// TIA Portal project "Nauriz_uploaded" (V17)

(* hardware
DEVICE "S7-1200 station_1"  S7-1200 Station
   slot 0: "Rack_0"  S7-1200 Rack  Rack  V1.0
   slot 1: "PLC_1"  CPU 1214C DC/DC/DC  6ES7 214-1AG40-0XB0  V4.4
   slot 2: "DI 16x24VDC/DQ 16xRelay_1"  SM 1223 DI16/DQ16 x relay  6ES7 223-1PL32-0XB0  V2.0
   slot 3: "DI 16/DQ 16x24VDC_1"  6ES7 223-1BL32-0XB0  V2.0
   slot 4: "DI 16x24VDC_1"  6ES7 221-1BH32-0XB0  V2.0
   slot 5: "DI 16x24VDC_2"  6ES7 221-1BH32-0XB0  V2.0
   slot 6: "AI 8x13BIT_1"  6ES7 231-4HF32-0XB0  V2.1
   slot 7: "AI 4x13BIT_1"  6ES7 231-4HD32-0XB0  V2.1
   slot 101: "CM 1241 (RS422/485)_1"  6ES7 241-1CH32-0XB0  V2.2
*)

// ===== PLC "PLC_1"  CPU 1214C DC/DC/DC =====

VAR_GLOBAL   // PLC tag table "Default tag table"
   "DIa1.0" AT %I0.0 : Bool;   // Наличие напряжения на основном вводе
   "DIa1.1" AT %I0.1 : Bool;   // Наличие напряжения на резервном вводе
   "DIa1.2" AT %I0.2 : Bool;   // Наличие питания 220 внешних потребителей
   "DIa1.3" AT %I0.3 : Bool;   // Наличие питания 220 собственных нужд
   "DIa1.4" AT %I0.4 : Bool;   // Отключение звука
   "DIa1.5" AT %I0.5 : Bool;   // Стоп АН
   "DIa1.6" AT %I0.6 : Bool;   // Автоматическое управление
   "DIa1.7" AT %I0.7 : Bool;   // Ручное управление
   "DIb1.0" AT %I1.0 : Bool;   // Тест индикации
   "DIb1.1" AT %I1.1 : Bool;   // Затопление
   "DIb1.2" AT %I1.2 : Bool;   // Открытие двери
   "Reserved DIb1.3" AT %I1.3 : Bool;   // ------------------------
   "Reserved DIb1.4" AT %I1.4 : Bool;   // ------------------------
   "Reserved DIb1.5" AT %I1.5 : Bool;   // ------------------------
   "DIa2.0" AT %I8.0 : Bool;   // Авт. выкл. НБ1 включен
   "DIa2.1" AT %I8.1 : Bool;   // Контактор НБ1 включен
   "DIa2.2" AT %I8.2 : Bool;   // Авт. выкл. НБ2 включен
   "DIa2.3" AT %I8.3 : Bool;   // Контактор НБ2 включен
   "DIa2.4" AT %I8.4 : Bool;   // Авт. выкл. НБ3 включен
   "DIa2.5" AT %I8.5 : Bool;   // Контактор НБ3 включен
   "DIa2.6" AT %I8.6 : Bool;   // Авт. выкл. НБ4 включен
   "DIa2.7" AT %I8.7 : Bool;   // Контактор НБ4 включен
   "DIb2.0" AT %I9.0 : Bool;   // Авт. выкл. НБ5 включен
   "DIb2.1" AT %I9.1 : Bool;   // Контактор НБ5 включен
   "DIb2.2" AT %I9.2 : Bool;   // Авт. выкл. НП включен
   "DIb2.3" AT %I9.3 : Bool;   // Контактор НП включен
   "DIb2.4" AT %I9.4 : Bool;   // Авт. выкл. ДР.Н включен
   "DIb2.5" AT %I9.5 : Bool;   // Контактор ДР.Н включен
   "Reserved DIb2.6" AT %I9.6 : Bool;   // ------------------------
   "Reserved DIb2.7" AT %I9.7 : Bool;   // ------------------------
   "DIa3.0" AT %I12.0 : Bool;   // УУС1: Проток
   "DIa3.1" AT %I12.1 : Bool;   // УУС2: Проток
   "DIa3.2" AT %I12.2 : Bool;   // УУС3: Проток
   "DIa3.3" AT %I12.3 : Bool;   // УУС4: Проток
   "DIa3.4" AT %I12.4 : Bool;   // УУС5: Проток
   "DIa3.5" AT %I12.5 : Bool;   // СПЖ1: Проток
   "DIa3.6" AT %I12.6 : Bool;   // Кнопка: Открыть УУД1
   "DIa3.7" AT %I12.7 : Bool;   // АПС: Открыть УУД1
   "DIb3.0" AT %I13.0 : Bool;   // УУС1: Открыт
   "DIb3.1" AT %I13.1 : Bool;   // УУС2: Открыт
   "DIb3.2" AT %I13.2 : Bool;   // УУС3: Открыт
   "DIb3.3" AT %I13.3 : Bool;   // УУС4: Открыт
   "DIb3.4" AT %I13.4 : Bool;   // УУС5: Открыт
   "Reserved DIb3.5" AT %I13.5 : Bool;   // ------------------------
   "Reserved DIb3.6" AT %I13.6 : Bool;   // ------------------------
   "Reserved DIb3.7" AT %I13.7 : Bool;   // ------------------------
   "DIa4.0" AT %I16.0 : Bool;   // Пож. резервуар: Уровень 1
   "DIa4.1" AT %I16.1 : Bool;   // Пож. резервуар: Уровень 2
   "DIa4.2" AT %I16.2 : Bool;   // Пож. резервуар: Уровень 3
   "DIa4.3" AT %I16.3 : Bool;   // Др. приямок: Вкл. ДР.Н
   "DIa4.4" AT %I16.4 : Bool;   // Др. приямок: Верх
   "Reserved DIa4.5" AT %I16.5 : Bool;   // ------------------------
   "Reserved DIa4.6" AT %I16.6 : Bool;   // ------------------------
   "Reserved DIa4.7" AT %I16.7 : Bool;   // ------------------------
   "Reserved DIb4.0" AT %I17.0 : Bool;   // ------------------------
   "Reserved DIb4.1" AT %I17.1 : Bool;   // ------------------------
   "DIb4.2" AT %I17.2 : Bool;   // КР.Ш38 УУС1: Открыт
   "DIb4.3" AT %I17.3 : Bool;   // КР.Ш38 УУС2: Открыт
   "DIb4.4" AT %I17.4 : Bool;   // КР.Ш38 УУС3: Открыт
   "DIb4.5" AT %I17.5 : Bool;   // КР.Ш38 УУС4: Открыт
   "DIb4.6" AT %I17.6 : Bool;   // КР.Ш38 УУС5: Открыт
   "DIb4.7" AT %I17.7 : Bool;   // КР.Ш38 УУД1: Открыт
   "DIa5.0" AT %I20.0 : Bool;   // КР.Ш12 УУС1: Открыт
   "DIa5.1" AT %I20.1 : Bool;   // КР.Ш12 УУС2: Открыт
   "DIa5.2" AT %I20.2 : Bool;   // КР.Ш12 УУС3: Открыт
   "DIa5.3" AT %I20.3 : Bool;   // КР.Ш12 УУС4: Открыт
   "DIa5.4" AT %I20.4 : Bool;   // КР.Ш12 УУС5: Открыт
   "Reserved DIa5.5" AT %I20.5 : Bool;   // ------------------------
   "Reserved DIa5.6" AT %I20.6 : Bool;   // ------------------------
   "Reserved DIa5.7" AT %I20.7 : Bool;   // ------------------------
   "Reserved DIb5.0" AT %I21.0 : Bool;   // ------------------------
   "Reserved DIb5.1" AT %I21.1 : Bool;   // ------------------------
   "Reserved DIb5.2" AT %I21.2 : Bool;   // ------------------------
   "Reserved DIb5.3" AT %I21.3 : Bool;   // ------------------------
   "Reserved DIb5.4" AT %I21.4 : Bool;   // ------------------------
   "Reserved DIb5.5" AT %I21.5 : Bool;   // ------------------------
   "Reserved DIb5.6" AT %I21.6 : Bool;   // ------------------------
   "Reserved DIb5.7" AT %I21.7 : Bool;   // ------------------------
   "AI6.0" AT %IW160 : Int;   // Датчик низкого давления PIS1.1
   "AI6.1" AT %IW162 : Int;   // Датчик низкого давления PIS1.2
   "AI6.2" AT %IW164 : Int;   // Датчик высокого давления PIS2.1
   "AI6.3" AT %IW166 : Int;   // Датчик высокого давления PIS2.2
   "AI6.4" AT %IW168 : Int;   // Датчик давления НБ1
   "AI6.5" AT %IW170 : Int;   // Датчик давления НБ2
   "AI6.6" AT %IW172 : Int;   // Датчик давления НБ3
   "AI6.7" AT %IW174 : Int;   // Датчик давления НБ4
   "AI7.0" AT %IW176 : Int;   // Датчик давления НБ5
   "AI7.1" AT %IW178 : Int;   // Датчик давления УУД1
   "Reserved AI7.2" AT %IW180 : Int;   // ------------------------
   "Reserved AI7.3" AT %IW182 : Int;   // ------------------------
   "DQa1.0" AT %Q0.0 : Bool;   // Пожар
   "DQa1.1" AT %Q0.1 : Bool;   // Пуск
   "DQa1.2" AT %Q0.2 : Bool;   // Неисправность
   "DQa1.3" AT %Q0.3 : Bool;   // Автоматика отключена
   "DQa1.4" AT %Q0.4 : Bool;   // Дежурный режим
   "DQa1.5" AT %Q0.5 : Bool;   // Звуковой сигнал
   "DQa1.6" AT %Q0.6 : Bool;   // СИстема отключена
   "DQa1.7" AT %Q0.7 : Bool;   // Звук отключен
   "DQb1.0" AT %Q1.0 : Bool;   // Наличие ОТВ
   "Reserved DQb1.1" AT %Q1.1 : Bool;   // ------------------------
   "RQa2.0" AT %Q8.0 : Bool;   // Управление НБ1
   "RQa2.1" AT %Q8.1 : Bool;   // Управление НБ2
   "RQa2.2" AT %Q8.2 : Bool;   // Управление НБ3
   "RQa2.3" AT %Q8.3 : Bool;   // Управление НБ4
   "RQa2.4" AT %Q8.4 : Bool;   // Управление НБ5
   "RQa2.5" AT %Q8.5 : Bool;   // Управление НП
   "RQa2.6" AT %Q8.6 : Bool;   // Управление ДР.Н
   "RQa2.7" AT %Q8.7 : Bool;   // Управление УУД1
   "RQb2.0" AT %Q9.0 : Bool;   // Неисправность НБ1
   "RQb2.1" AT %Q9.1 : Bool;   // Неисправность НБ2
   "RQb2.2" AT %Q9.2 : Bool;   // Неисправность НБ3
   "RQb2.3" AT %Q9.3 : Bool;   // Неисправность НБ4
   "RQb2.4" AT %Q9.4 : Bool;   // Неисправность НБ5
   "RQb2.5" AT %Q9.5 : Bool;   // Неисправность НП
   "RQb2.6" AT %Q9.6 : Bool;   // Неисправность ДР.Н
   "Reserved RQb2.7" AT %Q9.7 : Bool;   // ------------------------
   "DQa3.0" AT %Q12.0 : Bool;   // УУС1: Срабатывание
   "DQa3.1" AT %Q12.1 : Bool;   // УУС1: Неисправность
   "DQa3.2" AT %Q12.2 : Bool;   // УУС2: Срабатывание
   "DQa3.3" AT %Q12.3 : Bool;   // УУС2: Неисправность
   "DQa3.4" AT %Q12.4 : Bool;   // УУС3: Срабатывание
   "DQa3.5" AT %Q12.5 : Bool;   // УУС3: Неисправность
   "DQa3.6" AT %Q12.6 : Bool;   // УУС4: Срабатывание
   "DQa3.7" AT %Q12.7 : Bool;   // УУС4: Неисправность
   "DQb3.0" AT %Q13.0 : Bool;   // УУС5: Срабатывание
   "DQb3.1" AT %Q13.1 : Bool;   // УУС5: Неисправность
   "DQb3.2" AT %Q13.2 : Bool;   // УУД1: Открыт
   "DQb3.3" AT %Q13.3 : Bool;   // УУД1: Неисправность
   "Reserved DQb3.4" AT %Q13.4 : Bool;   // ------------------------
   "Reserved DQb3.5" AT %Q13.5 : Bool;   // ------------------------
   "Reserved DQb3.6" AT %Q13.6 : Bool;   // ------------------------
   "Reserved DQb3.7" AT %Q13.7 : Bool;   // ------------------------
   "System_Byte" AT %MB1 : Byte;
   "FirstScan" AT %M1.0 : Bool;
   "DiagStatusUpdate" AT %M1.1 : Bool;
   "AlwaysTRUE" AT %M1.2 : Bool;
   "AlwaysFALSE" AT %M1.3 : Bool;
   "MB_MODE_AUTO" AT %M4001.1 : Bool;
   "MB_MODE_MANUAL" AT %M4001.2 : Bool;
   "MB_MODE_BLOCKED" AT %M4001.3 : Bool;
   "MB_MODE_STANDBY" AT %M4001.4 : Bool;
   "MB_ERROR_ANY" AT %M4003.5 : Bool;
   "MB_ERROR_INLET_PRESSURE_LOW" AT %M4004.0 : Bool;
   "MB_ERROR_PUMP1" AT %M4004.1 : Bool;
   "MB_ERROR_PUMP2" AT %M4004.2 : Bool;
   "MB_ERROR_PUMP3" AT %M4004.3 : Bool;
   "MB_ERROR_PUMP4" AT %M4004.4 : Bool;
   "MB_ERROR_PUMP5" AT %M4004.5 : Bool;
   "MB_ERROR_PRESSURE_SENSOR_PUMP1" AT %M4004.6 : Bool;
   "MB_ERROR_PRESSURE_SENSOR_PUMP2" AT %M4004.7 : Bool;
   "MB_ERROR_PRESSURE_SENSOR_PUMP3" AT %M4005.0 : Bool;
   "MB_ERROR_PRESSURE_SENSOR_PUMP4" AT %M4005.1 : Bool;
   "MB_ERROR_PRESSURE_SENSOR_PUMP5" AT %M4005.2 : Bool;
   "MB_BUTTON_GLOBAL_STOP" AT %M4005.3 : Bool;
   "MB_ERROR_STANDBY_PUMP" AT %M4005.4 : Bool;
   "MB_SENSOR_FLOW_UUS1" AT %M4005.6 : Bool;
   "MB_SENSOR_FLOW_UUS2" AT %M4005.7 : Bool;
   "MB_SENSOR_FLOW_UUS3" AT %M4006.0 : Bool;
   "MB_SENSOR_FLOW_UUS4" AT %M4006.1 : Bool;
   "MB_SENSOR_FLOW_UUS5" AT %M4006.2 : Bool;
   "MB_SIGNAL_OPEN_UUS1" AT %M4006.3 : Bool;
   "MB_SIGNAL_OPEN_UUS2" AT %M4006.4 : Bool;
   "MB_SIGNAL_OPEN_UUS3" AT %M4006.5 : Bool;
   "MB_SIGNAL_OPEN_UUS4" AT %M4006.6 : Bool;
   "MB_SIGNAL_OPEN_UUS5" AT %M4006.7 : Bool;
   "MB_SENSOR_ERROR_UUS1" AT %M4007.0 : Bool;
   "MB_SENSOR_ERROR_UUS2" AT %M4007.1 : Bool;
   "MB_SENSOR_ERROR_UUS3" AT %M4007.2 : Bool;
   "MB_SENSOR_ERROR_UUS4" AT %M4007.3 : Bool;
   "MB_SENSOR_ERROR_UUS5" AT %M4007.4 : Bool;
   "MB_SENSOR_OPEN_KP38.1" AT %M4007.5 : Bool;
   "MB_SENSOR_OPEN_KP38.2" AT %M4007.6 : Bool;
   "MB_SENSOR_OPEN_KP38.3" AT %M4007.7 : Bool;
   "MB_SENSOR_OPEN_KP38.4" AT %M4008.0 : Bool;
   "MB_SENSOR_OPEN_KP38.5" AT %M4008.1 : Bool;
   "MB_SENSOR_OPEN_KP38.6" AT %M4008.2 : Bool;
   "MB_STATE_380_MAIN" AT %M4001.5 : Bool;
   "MB_STATE_380_BACKUP" AT %M4001.6 : Bool;
   "MB_STATE_220_INNER" AT %M4001.7 : Bool;
   "MB_STATE_220_OUTER" AT %M4002.0 : Bool;
   "MB_STATE_DOOR_OPENED" AT %M4002.1 : Bool;
   "MB_ERROR_UNDERWATER" AT %M4002.3 : Bool;
   "MB_ERROR_NO_WATER" AT %M4002.4 : Bool;
   "MB_ERROR_NO_WATER_FIRE" AT %M4002.5 : Bool;
   "MB_ERROR_GLOBAL" AT %M4003.1 : Bool;
   "MB_ERROR_UUS" AT %M4003.2 : Bool;
   "MB_ERROR_UUS_ANY" AT %M4003.3 : Bool;
   "MB_ERROR_PUMPS" AT %M4003.6 : Bool;
   "MB_ERROR_BALL_VALVE_ANY" AT %M4003.7 : Bool;
   "MB_SIGNAL_FIRE" AT %M4002.2 : Bool;
   "MB_SENSOR_PRESSURE_PUMP1" AT %MD4012 : Real;
   "MB_SENSOR_PRESSURE_PUMP2" AT %MD4016 : Real;
   "MB_SENSOR_PRESSURE_PUMP3" AT %MD4020 : Real;
   "MB_SENSOR_PRESSURE_PUMP4" AT %MD4024 : Real;
   "MB_SENSOR_PRESSURE_PUMP5" AT %MD4028 : Real;
   "MB_SENSOR_INDICATION_PRESSURE_LOW" AT %MD4032 : Real;
   "MB_SENSOR_INDICATION_PRESSURE_HIGH" AT %MD4036 : Real;
   "MB_STATE_WORK_PUMP1" AT %M4009.0 : Bool;
   "MB_STATE_WORK_PUMP2" AT %M4009.1 : Bool;
   "MB_STATE_WORK_PUMP3" AT %M4009.2 : Bool;
   "MB_STATE_WORK_PUMP4" AT %M4009.3 : Bool;
   "MB_STATE_WORK_PUMP5" AT %M4009.4 : Bool;
   "MB_STATE_WORK_STANDBY_PUMP" AT %M4009.5 : Bool;
   "MB_STATE_WORK_ANY_PUMP" AT %M4009.6 : Bool;
   "MB_ERROR_CONNECTION_LOST" AT %M4010.5 : Bool;
   "MB_BUTTON_START_KPPU" AT %M4000.2 : Bool;
   "MB_BUTTON_STOP_KPPU" AT %M4000.1 : Bool;
   "MB_BUTTON_UUD_OPEN_KPPU" AT %M4000.3 : Bool;
   "MB_WATER_LEVEL_FULL" AT %M4002.6 : Bool;
   "MB_SIGNAL_NEED_REPLENISH_1" AT %M4002.7 : Bool;
   "MB_SIGNAL_NEED_REPLENISH_2" AT %M4003.0 : Bool;
   "MB_ERROR_UUD1" AT %M4003.4 : Bool;
   "MB_ERROR_DRAIN_PUMP" AT %M4005.5 : Bool;
   "MB_STATE_WORK_DRAIN_PUMP" AT %M4009.7 : Bool;
   "MB_Sensor_water_level_1" AT %M4010.0 : Bool;
   "MB_Sensor_water_level_2" AT %M4010.1 : Bool;
   "MB_Sensor_water_level_3" AT %M4010.2 : Bool;
   "MB_Sensor_drain_work" AT %M4010.3 : Bool;
   "MB_Sensor_drain_overflow" AT %M4010.4 : Bool;
   "MB_SENSOR_OPEN_KP12.1" AT %M4008.3 : Bool;
   "MB_SENSOR_OPEN_KP12.2" AT %M4008.4 : Bool;
   "MB_SENSOR_OPEN_KP12.3" AT %M4008.5 : Bool;
   "MB_SENSOR_OPEN_KP12.4" AT %M4008.6 : Bool;
   "MB_SENSOR_OPEN_KP12.5" AT %M4008.7 : Bool;
   "Commload_done" AT %M900.0 : Bool;
   "Master_reading_done" AT %M900.1 : Bool;
   "Master_writing_done" AT %M900.2 : Bool;
   "Master_reading_error" AT %M900.3 : Bool;
   "Master_writing_error" AT %M900.4 : Bool;
   "Master_read" AT %M900.5 : Bool;
   "Master_write" AT %M900.6 : Bool;
   "Error_connection_lost" AT %M900.7 : Bool;
   "WriteHoldingRegister_00" AT %MW4002 : Word;
   "WriteHoldingRegister_01" AT %MW4004 : Word;
   "WriteHoldingRegister_02" AT %MW4006 : Word;
   "WriteHoldingRegister_03" AT %MW4008 : Word;
   "WriteHoldingRegister_04" AT %MW4010 : Word;
   "WriteHoldingRegister_05" AT %MW4012 : Word;
   "WriteHoldingRegister_06" AT %MW4014 : Word;
   "WriteHoldingRegister_07" AT %MW4016 : Word;
   "WriteHoldingRegister_08" AT %MW4018 : Word;
   "WriteHoldingRegister_09" AT %MW4020 : Word;
   "WriteHoldingRegister_10" AT %MW4022 : Word;
   "WriteHoldingRegister_11" AT %MW4024 : Word;
   "WriteHoldingRegister_12" AT %MW4026 : Word;
   "WriteHoldingRegister_13" AT %MW4028 : Word;
   "WriteHoldingRegister_14" AT %MW4030 : Word;
   "WriteHoldingRegister_15" AT %MW4032 : Word;
   "WriteHoldingRegister_16" AT %MW4034 : Word;
   "WriteHoldingRegister_18" AT %MW4038 : Word;
   "WriteHoldingRegister_19" AT %MW4040 : Word;
   "WriteHoldingRegister_20" AT %MW4042 : Word;
   "WriteHoldingRegister_22" AT %MW4046 : Word;
   "WriteHoldingRegister_23" AT %MW4048 : Word;
   "WriteHoldingRegister_24" AT %MW4050 : Word;
   "WriteHoldingRegister_25" AT %MW4052 : Word;
   "WriteHoldingRegister_26" AT %MW4054 : Word;
   "WriteHoldingRegister_27" AT %MW4056 : Word;
   "WriteHoldingRegister_28" AT %MW4058 : Word;
   "WriteHoldingRegister_29" AT %MW4060 : Word;
   "WriteHoldingRegister_30" AT %MW4062 : Word;
   "WriteHoldingRegister_31" AT %MW4064 : Word;
   "WriteHoldingRegister_32" AT %MW4066 : Word;
   "WriteHoldingRegister_33" AT %MW4068 : Word;
   "WriteHoldingRegister_34" AT %MW4070 : Word;
   "WriteHoldingRegister_35" AT %MW4072 : Word;
   "WriteHoldingRegister_36" AT %MW4074 : Word;
   "WriteHoldingRegister_37" AT %MW4076 : Word;
   "WriteHoldingRegister_38" AT %MW4078 : Word;
   "ReadHolding" AT %MW4000 : Word;
   "WriteHoldingRegister_17" AT %MW4036 : Word;
   "WriteHoldingRegister_21" AT %MW4044 : Word;
   "HMI_MODE_AUTO" AT %M600.0 : Bool;
   "HMI_MODE_MANUAL" AT %M600.1 : Bool;
   "HMI_MODE_BLOCKED" AT %M600.2 : Bool;
   "HMI_MODE_STANDBY" AT %M600.3 : Bool;
   "HMI_ERROR_ANY" AT %M600.4 : Bool;
   "HMI_ERROR_INLET_PRESSURE_LOW" AT %M600.5 : Bool;
   "HMI_ERROR_PUMP1" AT %M600.6 : Bool;
   "HMI_ERROR_PUMP2" AT %M600.7 : Bool;
   "HMI_ERROR_PUMP3" AT %M601.0 : Bool;
   "HMI_ERROR_PUMP4" AT %M601.1 : Bool;
   "HMI_ERROR_PUMP5" AT %M601.2 : Bool;
   "HMI_ERROR_PRESSURE_SENSOR_PUMP1" AT %M601.3 : Bool;
   "HMI_ERROR_PRESSURE_SENSOR_PUMP2" AT %M601.4 : Bool;
   "HMI_ERROR_PRESSURE_SENSOR_PUMP3" AT %M601.5 : Bool;
   "HMI_ERROR_PRESSURE_SENSOR_PUMP4" AT %M601.6 : Bool;
   "HMI_ERROR_PRESSURE_SENSOR_PUMP5" AT %M601.7 : Bool;
   "HMI_BUTTON_GLOBAL_STOP" AT %M602.0 : Bool;
   "HMI_ERROR_STANDBY_PUMP" AT %M602.1 : Bool;
   "HMI_SENSOR_FLOW_UUS1" AT %M602.2 : Bool;
   "HMI_SENSOR_FLOW_UUS2" AT %M602.3 : Bool;
   "HMI_SENSOR_FLOW_UUS3" AT %M602.4 : Bool;
   "HMI_SENSOR_FLOW_UUS4" AT %M602.5 : Bool;
   "HMI_SENSOR_FLOW_UUS5" AT %M602.6 : Bool;
   "HMI_SIGNAL_OPEN_UUS1" AT %M602.7 : Bool;
   "HMI_SIGNAL_OPEN_UUS2" AT %M603.0 : Bool;
   "HMI_SIGNAL_OPEN_UUS3" AT %M603.1 : Bool;
   "HMI_SIGNAL_OPEN_UUS4" AT %M603.2 : Bool;
   "HMI_SIGNAL_OPEN_UUS5" AT %M603.3 : Bool;
   "HMI_SENSOR_ERROR_UUS1" AT %M603.4 : Bool;
   "HMI_SENSOR_ERROR_UUS2" AT %M603.5 : Bool;
   "HMI_SENSOR_ERROR_UUS3" AT %M603.6 : Bool;
   "HMI_SENSOR_ERROR_UUS4" AT %M603.7 : Bool;
   "HMI_SENSOR_ERROR_UUS5" AT %M604.0 : Bool;
   "HMI_SENSOR_OPEN_KP38.1" AT %M604.1 : Bool;
   "HMI_SENSOR_OPEN_KP38.2" AT %M604.2 : Bool;
   "HMI_SENSOR_OPEN_KP38.3" AT %M604.3 : Bool;
   "HMI_SENSOR_OPEN_KP38.4" AT %M604.4 : Bool;
   "HMI_SENSOR_OPEN_KP38.5" AT %M604.5 : Bool;
   "HMI_SENSOR_OPEN_KP38.6" AT %M604.6 : Bool;
   "HMI_STATE_380_MAIN" AT %M604.7 : Bool;
   "HMI_STATE_380_BACKUP" AT %M605.0 : Bool;
   "HMI_STATE_220_INNER" AT %M605.1 : Bool;
   "HMI_STATE_220_OUTER" AT %M605.2 : Bool;
   "HMI_STATE_DOOR_OPENED" AT %M605.3 : Bool;
   "HMI_ERROR_UNDERWATER" AT %M605.4 : Bool;
   "HMI_ERROR_NO_WATER" AT %M605.5 : Bool;
   "HMI_ERROR_NO_WATER_FIRE" AT %M605.6 : Bool;
   "HMI_ERROR_GLOBAL" AT %M605.7 : Bool;
   "HMI_ERROR_UUS" AT %M606.0 : Bool;
   "HMI_ERROR_UUS_ANY" AT %M606.1 : Bool;
   "HMI_ERROR_PUMPS" AT %M606.2 : Bool;
   "HMI_ERROR_BALL_VALVE_ANY" AT %M606.3 : Bool;
   "HMI_SIGNAL_FIRE" AT %M606.4 : Bool;
   "HMI_SENSOR_PRESSURE_PUMP1" AT %MD610 : Real;
   "HMI_SENSOR_PRESSURE_PUMP2" AT %MD614 : Real;
   "HMI_SENSOR_PRESSURE_PUMP3" AT %MD618 : Real;
   "HMI_SENSOR_PRESSURE_PUMP4" AT %MD622 : Real;
   "HMI_SENSOR_PRESSURE_PUMP5" AT %MD626 : Real;
   "HMI_SENSOR_INDICATION_PRESSURE_LOW" AT %MD630 : Real;
   "HMI_SENSOR_INDICATION_PRESSURE_HIGH" AT %MD634 : Real;
   "HMI_STATE_WORK_PUMP1" AT %M606.5 : Bool;
   "HMI_STATE_WORK_PUMP2" AT %M606.6 : Bool;
   "HMI_STATE_WORK_PUMP3" AT %M606.7 : Bool;
   "HMI_STATE_WORK_PUMP4" AT %M607.0 : Bool;
   "HMI_STATE_WORK_PUMP5" AT %M607.1 : Bool;
   "HMI_STATE_WORK_STANDBY_PUMP" AT %M607.2 : Bool;
   "HMI_STATE_WORK_ANY_PUMP" AT %M607.3 : Bool;
   "HMI_ERROR_CONNECTION_LOST" AT %M607.4 : Bool;
   "HMI_BUTTON_START_KPPU" AT %M607.5 : Bool;
   "HMI_BUTTON_STOP_KPPU" AT %M607.6 : Bool;
   "HMI_BUTTON_UUD_OPEN_KPPU" AT %M607.7 : Bool;
   "HMI_WATER_LEVEL_FULL" AT %M608.0 : Bool;
   "HMI_SIGNAL_NEED_REPLENISH_1" AT %M608.1 : Bool;
   "HMI_SIGNAL_NEED_REPLENISH_2" AT %M608.2 : Bool;
   "HMI_ERROR_UUD1" AT %M608.3 : Bool;
   "HMI_ERROR_DRAIN_PUMP" AT %M608.4 : Bool;
   "HMI_STATE_WORK_DRAIN_PUMP" AT %M608.5 : Bool;
   "HMI_Sensor_water_level_1" AT %M608.6 : Bool;
   "HMI_Sensor_water_level_2" AT %M608.7 : Bool;
   "HMI_Sensor_water_level_3" AT %M609.0 : Bool;
   "HMI_Sensor_drain_work" AT %M609.1 : Bool;
   "HMI_Sensor_drain_overflow" AT %M609.2 : Bool;
   "HMI_SENSOR_OPEN_KP12.1" AT %M609.3 : Bool;
   "HMI_SENSOR_OPEN_KP12.2" AT %M609.4 : Bool;
   "HMI_SENSOR_OPEN_KP12.3" AT %M609.5 : Bool;
   "HMI_SENSOR_OPEN_KP12.4" AT %M609.6 : Bool;
   "HMI_SENSOR_OPEN_KP12.5" AT %M609.7 : Bool;
END_VAR

DATA_BLOCK "Ball_valves_data"   // DB1
{ S7_Optimized_Access := 'TRUE' }
VERSION : 0.1
   VAR
      SENSOR_KR38_open : Array[1..6] of Bool;
      SENSOR_KR12_open : Array[1..5] of Bool;
      SENSOR_ERROR_KR38 : Array[1..6] of Bool;
   END_VAR
BEGIN
END_DATA_BLOCK

DATA_BLOCK "Section_valves_data"   // DB2
{ S7_Optimized_Access := 'TRUE' }
VERSION : 0.1
   VAR
      SENSOR_flow_UUS : Array[1..5] of Bool;
      SENSOR_ERROR_UUS : Array[1..5] of Bool;
      SENSOR_open_UUS : Array[1..5] of Bool;
      SENSOR_ERROR_UUD1 : Bool;
      SENSOR_open_UUD1 : Bool;
      SENSOR_FALSE_UUD1 : Bool;
   END_VAR
BEGIN
END_DATA_BLOCK

DATA_BLOCK "Global"   // DB47
{ S7_Optimized_Access := 'TRUE' }
VERSION : 0.1
   VAR
      MODE_auto : Bool;
      MODE_manual : Bool;
      MODE_blocked : Bool;
      MODE_standby : Bool;
      BUTTON_Global_Stop : Bool;
      BUTTON_Sound_Off : Bool;
      BUTTON_Led_Test : Bool;
      BUTTON_UUD1_Open : Bool;
      STATE_380_main : Bool;
      STATE_380_backup : Bool;
      STATE_220_inner : Bool;
      STATE_220_outer : Bool;
      STATE_door_opened : Bool;
      ERROR_underwater : Bool;
      ERROR_no_water : Bool;
      ERROR_no_water_fire : Bool;
      ERROR_global : Bool;
      ERROR_UUS : Bool;
      ERROR_UUS_any : Bool;
      ERROR_any : Bool;
      ERROR_PUMPS : Bool;
      SIGNAL_fire : Bool;
      "SENSOR_low_pressure_PIS1.1" : Real;
      "SENSOR_low_pressure_PIS1.2" : Real := 0.0;
      "SENSOR_high_pressure_PIS2.1" : Real := 0.0;
      "SENSOR_high_pressure_PIS2.2" : Real := 0.0;
      SENSOR_high_pressure_pump_1 : Real := 0.0;
      SENSOR_high_pressure_pump_2 : Real := 0.0;
      SENSOR_high_pressure_pump_3 : Real := 0.0;
      SENSOR_high_pressure_pump_4 : Real := 0.0;
      SENSOR_high_pressure_pump_5 : Real := 0.0;
      SENSOR_high_pressure_UUD1 : Real;
      INDICATION_low_pressure : Real := 0.0;
      INDICATION_high_pressure : Real := 0.0;
      ERROR_main_ball_valves : Bool;
      ERROR_ball_valve_any : Bool;
      ERROR_inlet_pressure_low : Bool;
      SIGNAL_first_pump_has_started : Bool;
      Start_standby_pump : Bool;
      Secret_condition : Bool := false;
      Sensor_water_level_1 : Bool;
      Sensor_water_level_2 : Bool;
      Sensor_water_level_3 : Bool;
      Sensor_drain_work : Bool;
      Sensor_drain_overflow : Bool;
      AI_sensors_error : Array[1..4] of Bool;
   END_VAR
BEGIN
END_DATA_BLOCK

DATA_BLOCK "AI_Sensor_high_pressure_UUD1"   // DB58
{ S7_Optimized_Access := 'TRUE' }
VERSION : 0.1
// stored: InstanceOfName AI_Sensor
"AI_Sensor"
BEGIN
END_DATA_BLOCK

DATA_BLOCK "Sound_DB"   // DB59
{ S7_Optimized_Access := 'TRUE' }
VERSION : 0.1
// stored: InstanceOfName Sound_PTO
"Sound_PTO"
BEGIN
END_DATA_BLOCK

DATA_BLOCK "Preset_values"   // DB69
{ S7_Optimized_Access := 'TRUE' }
VERSION : 0.1
   VAR
      DI_timer_delay_time_superfast : Time := T#0.2s;
      DI_timer_delay_time_fast : Time := T#0.5s;
      DI_timer_delay_time_regular : Time := T#1s;
      DI_timer_delay_time_slow : Time := T#3s;
      DI_timer_delay_time_superslow : Time := T#5s;
      DI_timer_delay_time_gate_valve : Time := T#30s;
      Pressure_stanby_low : Real := 2.29;
      Pressure_stanby_pump_on : Real := 2.3;
      Pressure_stanby_pump_stop : Real := 2.5;
      Pressure_cascade_start : Real := 7.5;
      Pressure_cascade_stop : Real := 9.0;
      Pressure_pump_is_ok : Real := 10.0;
      Timer_cascade_start : Time := T#25s;
      Pump_error_time_by_pressure : Time := T#60s;
   END_VAR
BEGIN
END_DATA_BLOCK

DATA_BLOCK "Water_control"   // DB71
{ S7_Optimized_Access := 'TRUE' }
VERSION : 0.1
   VAR
      Water_level_full : Bool;
      Signal_need_replenish_1 : Bool;
      Signal_need_replenish_2 : Bool;
   END_VAR
BEGIN
END_DATA_BLOCK

DATA_BLOCK "Cascade_start_stop_DB"   // DB72
{ S7_Optimized_Access := 'TRUE' }
VERSION : 0.1
// stored: InstanceOfName Cascade_start_stop
"Cascade_start_stop"
BEGIN
END_DATA_BLOCK

DATA_BLOCK "Pumps_data"   // DB73
{ S7_Optimized_Access := 'TRUE' }
VERSION : 0.1
   VAR
      State_switch_pump : Array[1..5] of Bool;
      Error_pump : Array[1..5] of Bool;
      State_starter_pump : Array[1..5] of Bool;
      State_work_pump : Array[1..5] of Bool;
      Pumps : Array[1..5] of Int;
      Pump_sensor_error : Array[1..5] of Bool;
      State_switch_standby_pump : Bool;
      Error_any_pump : Bool;
      Error_standby_pump : Bool;
      State_starter_standby_pump : Bool;
      State_work_standby_pump : Bool;
      State_work_any_pump : Bool;
      State_switch_drain_pump : Bool;
      State_starter_drain_pump : Bool;
      Error_drain_pump : Bool;
      State_work_drain_pump : Bool;
   END_VAR
BEGIN
END_DATA_BLOCK

DATA_BLOCK "Data_push_to_MODBUS_DB"   // DB85
{ S7_Optimized_Access := 'TRUE' }
VERSION : 0.1
// stored: InstanceOfName Data_push_to_MODBUS
"Data_push_to_MODBUS"
BEGIN
END_DATA_BLOCK

DATA_BLOCK "Data_push_to_HMI_DB"   // DB87
{ S7_Optimized_Access := 'TRUE' }
VERSION : 0.1
// stored: InstanceOfName Data_push_to_HMI
"Data_push_to_HMI"
BEGIN
END_DATA_BLOCK

DATA_BLOCK "User_Defined"   // DB100
{ S7_Optimized_Access := 'TRUE' }
VERSION : 0.1
   VAR
      Pressure_stanby_low : Real := 2.29;
      Pressure_stanby_pump_on : Real := 2.3;
      Pressure_stanby_pump_stop : Real := 2.5;
      Pressure_cascade_start : Real := 7.5;
      Pressure_cascade_stop : Real := 9.0;
      Pressure_pump_is_ok : Real := 10.0;
      Timer_cascade_start : Time := T#25s;
      Timer_standby_pump : Time := T#40ms;
      Pump_error_time_by_pressure : Time := T#60s;
   END_VAR
BEGIN
END_DATA_BLOCK

// folder: AI_db

DATA_BLOCK "AI_Sensor_low_pressure_PIS1.1"   // DB43
{ S7_Optimized_Access := 'TRUE' }
VERSION : 0.1
// stored: InstanceOfName AI_Sensor
"AI_Sensor"
BEGIN
END_DATA_BLOCK

DATA_BLOCK "AI_Sensor_low_pressure_PIS1.2"   // DB44
{ S7_Optimized_Access := 'TRUE' }
VERSION : 0.1
// stored: InstanceOfName AI_Sensor
"AI_Sensor"
BEGIN
END_DATA_BLOCK

DATA_BLOCK "AI_Sensor_high_pressure_PIS2.1"   // DB45
{ S7_Optimized_Access := 'TRUE' }
VERSION : 0.1
// stored: InstanceOfName AI_Sensor
"AI_Sensor"
BEGIN
END_DATA_BLOCK

DATA_BLOCK "AI_Sensor_high_pressure_PIS2.2"   // DB46
{ S7_Optimized_Access := 'TRUE' }
VERSION : 0.1
// stored: InstanceOfName AI_Sensor
"AI_Sensor"
BEGIN
END_DATA_BLOCK

DATA_BLOCK "AI_Sensor_high_pressure_pump_1"   // DB48
{ S7_Optimized_Access := 'TRUE' }
VERSION : 0.1
// stored: InstanceOfName AI_Sensor
"AI_Sensor"
BEGIN
END_DATA_BLOCK

DATA_BLOCK "AI_Sensor_high_pressure_pump_2"   // DB49
{ S7_Optimized_Access := 'TRUE' }
VERSION : 0.1
// stored: InstanceOfName AI_Sensor
"AI_Sensor"
BEGIN
END_DATA_BLOCK

DATA_BLOCK "AI_Sensor_high_pressure_pump_3"   // DB50
{ S7_Optimized_Access := 'TRUE' }
VERSION : 0.1
// stored: InstanceOfName AI_Sensor
"AI_Sensor"
BEGIN
END_DATA_BLOCK

DATA_BLOCK "AI_Sensor_high_pressure_pump_4"   // DB51
{ S7_Optimized_Access := 'TRUE' }
VERSION : 0.1
// stored: InstanceOfName AI_Sensor
"AI_Sensor"
BEGIN
END_DATA_BLOCK

DATA_BLOCK "AI_Sensor_high_pressure_pump_5"   // DB52
{ S7_Optimized_Access := 'TRUE' }
VERSION : 0.1
// stored: InstanceOfName AI_Sensor
"AI_Sensor"
BEGIN
END_DATA_BLOCK

DATA_BLOCK "AI_Redundancy_low_pressure"   // DB56
{ S7_Optimized_Access := 'TRUE' }
VERSION : 0.1
// stored: InstanceOfName AI_Redundancy
"AI_Redundancy"
BEGIN
END_DATA_BLOCK

DATA_BLOCK "AI_Redundancy_high_pressure"   // DB57
{ S7_Optimized_Access := 'TRUE' }
VERSION : 0.1
// stored: InstanceOfName AI_Redundancy
"AI_Redundancy"
BEGIN
END_DATA_BLOCK

// folder: DI_db

DATA_BLOCK "State_380_main"   // DB3
{ S7_Optimized_Access := 'TRUE' }
VERSION : 0.1
// stored: InstanceOfName DI_Single
"DI_Single"
BEGIN
END_DATA_BLOCK

DATA_BLOCK "State_380_backup"   // DB4
{ S7_Optimized_Access := 'TRUE' }
VERSION : 0.1
// stored: InstanceOfName DI_Single
"DI_Single"
BEGIN
END_DATA_BLOCK

DATA_BLOCK "State_220_outer"   // DB5
{ S7_Optimized_Access := 'TRUE' }
VERSION : 0.1
// stored: InstanceOfName DI_Single
"DI_Single"
BEGIN
END_DATA_BLOCK

DATA_BLOCK "State_220_inner"   // DB6
{ S7_Optimized_Access := 'TRUE' }
VERSION : 0.1
// stored: InstanceOfName DI_Single
"DI_Single"
BEGIN
END_DATA_BLOCK

DATA_BLOCK "State_Mode_Auto"   // DB7
{ S7_Optimized_Access := 'TRUE' }
VERSION : 0.1
// stored: InstanceOfName DI_Single
"DI_Single"
BEGIN
END_DATA_BLOCK

DATA_BLOCK "State_mode_manual"   // DB8
{ S7_Optimized_Access := 'TRUE' }
VERSION : 0.1
// stored: InstanceOfName DI_Single
"DI_Single"
BEGIN
END_DATA_BLOCK

DATA_BLOCK "State_underwater"   // DB9
{ S7_Optimized_Access := 'TRUE' }
VERSION : 0.1
// stored: InstanceOfName DI_Single
"DI_Single"
BEGIN
END_DATA_BLOCK

DATA_BLOCK "State_door_opened"   // DB10
{ S7_Optimized_Access := 'TRUE' }
VERSION : 0.1
// stored: InstanceOfName DI_Single
"DI_Single"
BEGIN
END_DATA_BLOCK

DATA_BLOCK "Button_UUD1_Open"   // DB11
{ S7_Optimized_Access := 'TRUE' }
VERSION : 0.1
// stored: InstanceOfName DI_Single
"DI_Single"
BEGIN
END_DATA_BLOCK

DATA_BLOCK "Button_sound_off"   // DB12
{ S7_Optimized_Access := 'TRUE' }
VERSION : 0.1
// stored: InstanceOfName DI_Single
"DI_Single"
BEGIN
END_DATA_BLOCK

DATA_BLOCK "Button_global_stop"   // DB13
{ S7_Optimized_Access := 'TRUE' }
VERSION : 0.1
// stored: InstanceOfName DI_Single
"DI_Single"
BEGIN
END_DATA_BLOCK

DATA_BLOCK "Button_led_test"   // DB14
{ S7_Optimized_Access := 'TRUE' }
VERSION : 0.1
// stored: InstanceOfName DI_Single
"DI_Single"
BEGIN
END_DATA_BLOCK

DATA_BLOCK "State_pump_1"   // DB15
{ S7_Optimized_Access := 'TRUE' }
VERSION : 0.1
// stored: InstanceOfName DI_Single
"DI_Single"
BEGIN
END_DATA_BLOCK

DATA_BLOCK "State_pump_2"   // DB16
{ S7_Optimized_Access := 'TRUE' }
VERSION : 0.1
// stored: InstanceOfName DI_Single
"DI_Single"
BEGIN
END_DATA_BLOCK

DATA_BLOCK "State_pump_3"   // DB17
{ S7_Optimized_Access := 'TRUE' }
VERSION : 0.1
// stored: InstanceOfName DI_Single
"DI_Single"
BEGIN
END_DATA_BLOCK

DATA_BLOCK "State_pump_4"   // DB18
{ S7_Optimized_Access := 'TRUE' }
VERSION : 0.1
// stored: InstanceOfName DI_Single
"DI_Single"
BEGIN
END_DATA_BLOCK

DATA_BLOCK "State_pump_5"   // DB19
{ S7_Optimized_Access := 'TRUE' }
VERSION : 0.1
// stored: InstanceOfName DI_Single
"DI_Single"
BEGIN
END_DATA_BLOCK

DATA_BLOCK "State_drain_pump"   // DB20
{ S7_Optimized_Access := 'TRUE' }
VERSION : 0.1
// stored: InstanceOfName DI_Single
"DI_Single"
BEGIN
END_DATA_BLOCK

DATA_BLOCK "State_starter_drain_pump"   // DB21
{ S7_Optimized_Access := 'TRUE' }
VERSION : 0.1
// stored: InstanceOfName DI_Single
"DI_Single"
BEGIN
END_DATA_BLOCK

DATA_BLOCK "Sensor_UUS1_Open"   // DB22
{ S7_Optimized_Access := 'TRUE' }
VERSION : 0.1
// stored: InstanceOfName DI_Single
"DI_Single"
BEGIN
END_DATA_BLOCK

DATA_BLOCK "State_standby_pump"   // DB23
{ S7_Optimized_Access := 'TRUE' }
VERSION : 0.1
// stored: InstanceOfName DI_Single
"DI_Single"
BEGIN
END_DATA_BLOCK

DATA_BLOCK "State_starter_pump_1"   // DB24
{ S7_Optimized_Access := 'TRUE' }
VERSION : 0.1
// stored: InstanceOfName DI_Single
"DI_Single"
BEGIN
END_DATA_BLOCK

DATA_BLOCK "State_starter_pump_2"   // DB25
{ S7_Optimized_Access := 'TRUE' }
VERSION : 0.1
// stored: InstanceOfName DI_Single
"DI_Single"
BEGIN
END_DATA_BLOCK

DATA_BLOCK "State_starter_pump_3"   // DB26
{ S7_Optimized_Access := 'TRUE' }
VERSION : 0.1
// stored: InstanceOfName DI_Single
"DI_Single"
BEGIN
END_DATA_BLOCK

DATA_BLOCK "State_starter_pump_4"   // DB27
{ S7_Optimized_Access := 'TRUE' }
VERSION : 0.1
// stored: InstanceOfName DI_Single
"DI_Single"
BEGIN
END_DATA_BLOCK

DATA_BLOCK "State_starter_pump_5"   // DB28
{ S7_Optimized_Access := 'TRUE' }
VERSION : 0.1
// stored: InstanceOfName DI_Single
"DI_Single"
BEGIN
END_DATA_BLOCK

DATA_BLOCK "Sensor_UUS2_open"   // DB29
{ S7_Optimized_Access := 'TRUE' }
VERSION : 0.1
// stored: InstanceOfName DI_Single
"DI_Single"
BEGIN
END_DATA_BLOCK

DATA_BLOCK "Sensor_UUS3_open"   // DB30
{ S7_Optimized_Access := 'TRUE' }
VERSION : 0.1
// stored: InstanceOfName DI_Single
"DI_Single"
BEGIN
END_DATA_BLOCK

DATA_BLOCK "Sensor_UUS4_open"   // DB31
{ S7_Optimized_Access := 'TRUE' }
VERSION : 0.1
// stored: InstanceOfName DI_Single
"DI_Single"
BEGIN
END_DATA_BLOCK

DATA_BLOCK "State_starter_standby_pump"   // DB32
{ S7_Optimized_Access := 'TRUE' }
VERSION : 0.1
// stored: InstanceOfName DI_Single
"DI_Single"
BEGIN
END_DATA_BLOCK

DATA_BLOCK "Sensor_flow_UUS1"   // DB33
{ S7_Optimized_Access := 'TRUE' }
VERSION : 0.1
// stored: InstanceOfName DI_Single
"DI_Single"
BEGIN
END_DATA_BLOCK

DATA_BLOCK "Sensor_flow_UUS2"   // DB34
{ S7_Optimized_Access := 'TRUE' }
VERSION : 0.1
// stored: InstanceOfName DI_Single
"DI_Single"
BEGIN
END_DATA_BLOCK

DATA_BLOCK "Sensor_flow_UUS3"   // DB35
{ S7_Optimized_Access := 'TRUE' }
VERSION : 0.1
// stored: InstanceOfName DI_Single
"DI_Single"
BEGIN
END_DATA_BLOCK

DATA_BLOCK "Sensor_flow_UUS4"   // DB36
{ S7_Optimized_Access := 'TRUE' }
VERSION : 0.1
// stored: InstanceOfName DI_Single
"DI_Single"
BEGIN
END_DATA_BLOCK

DATA_BLOCK "Sensor_flow_UUS5"   // DB37
{ S7_Optimized_Access := 'TRUE' }
VERSION : 0.1
// stored: InstanceOfName DI_Single
"DI_Single"
BEGIN
END_DATA_BLOCK

DATA_BLOCK "Sensor_UUS5_open"   // DB38
{ S7_Optimized_Access := 'TRUE' }
VERSION : 0.1
// stored: InstanceOfName DI_Single
"DI_Single"
BEGIN
END_DATA_BLOCK

DATA_BLOCK "Sensor_KR38.1_open"   // DB39
{ S7_Optimized_Access := 'TRUE' }
VERSION : 0.1
// stored: InstanceOfName DI_Single
"DI_Single"
BEGIN
END_DATA_BLOCK

DATA_BLOCK "Sensor_KR38.2_open"   // DB40
{ S7_Optimized_Access := 'TRUE' }
VERSION : 0.1
// stored: InstanceOfName DI_Single
"DI_Single"
BEGIN
END_DATA_BLOCK

DATA_BLOCK "Sensor_KR38.3_open"   // DB41
{ S7_Optimized_Access := 'TRUE' }
VERSION : 0.1
// stored: InstanceOfName DI_Single
"DI_Single"
BEGIN
END_DATA_BLOCK

DATA_BLOCK "Sensor_KR38.4_open"   // DB42
{ S7_Optimized_Access := 'TRUE' }
VERSION : 0.1
// stored: InstanceOfName DI_Single
"DI_Single"
BEGIN
END_DATA_BLOCK

DATA_BLOCK "Sensor_water_level_3"   // DB53
{ S7_Optimized_Access := 'TRUE' }
VERSION : 0.1
// stored: InstanceOfName DI_Single
"DI_Single"
BEGIN
END_DATA_BLOCK

DATA_BLOCK "Sensor_drain_work"   // DB54
{ S7_Optimized_Access := 'TRUE' }
VERSION : 0.1
// stored: InstanceOfName DI_Single
"DI_Single"
BEGIN
END_DATA_BLOCK

DATA_BLOCK "Sensor_drain_overflow"   // DB55
{ S7_Optimized_Access := 'TRUE' }
VERSION : 0.1
// stored: InstanceOfName DI_Single
"DI_Single"
BEGIN
END_DATA_BLOCK

DATA_BLOCK "Standby_Pump/Compressor_Error_DB"   // DB60
{ S7_Optimized_Access := 'TRUE' }
VERSION : 0.1
// stored: InstanceOfName Standby_Pump/Compressor_Error
"Standby_Pump/Compressor_Error"
BEGIN
END_DATA_BLOCK

DATA_BLOCK "Pump_Error_1"   // DB61
{ S7_Optimized_Access := 'TRUE' }
VERSION : 0.1
// stored: InstanceOfName Pump_Error
"Pump_Error"
BEGIN
END_DATA_BLOCK

DATA_BLOCK "Pump_Error_2"   // DB62
{ S7_Optimized_Access := 'TRUE' }
VERSION : 0.1
// stored: InstanceOfName Pump_Error
"Pump_Error"
BEGIN
END_DATA_BLOCK

DATA_BLOCK "Pump_Error_3"   // DB63
{ S7_Optimized_Access := 'TRUE' }
VERSION : 0.1
// stored: InstanceOfName Pump_Error
"Pump_Error"
BEGIN
END_DATA_BLOCK

DATA_BLOCK "Pump_Error_4"   // DB64
{ S7_Optimized_Access := 'TRUE' }
VERSION : 0.1
// stored: InstanceOfName Pump_Error
"Pump_Error"
BEGIN
END_DATA_BLOCK

DATA_BLOCK "Pump_Error_5"   // DB65
{ S7_Optimized_Access := 'TRUE' }
VERSION : 0.1
// stored: InstanceOfName Pump_Error
"Pump_Error"
BEGIN
END_DATA_BLOCK

DATA_BLOCK "Drain_pump_error"   // DB66
{ S7_Optimized_Access := 'TRUE' }
VERSION : 0.1
// stored: InstanceOfName Standby_Pump/Compressor_Error
"Standby_Pump/Compressor_Error"
BEGIN
END_DATA_BLOCK

DATA_BLOCK "Button_open UUD_1"   // DB67
{ S7_Optimized_Access := 'TRUE' }
VERSION : 0.1
// stored: InstanceOfName Button_open UUD
"Button_open UUD"
BEGIN
END_DATA_BLOCK

DATA_BLOCK "Sensor_KR12.1_open"   // DB76
{ S7_Optimized_Access := 'TRUE' }
VERSION : 0.1
// stored: InstanceOfName DI_Single
"DI_Single"
BEGIN
END_DATA_BLOCK

DATA_BLOCK "Sensor_KR12.2_open"   // DB77
{ S7_Optimized_Access := 'TRUE' }
VERSION : 0.1
// stored: InstanceOfName DI_Single
"DI_Single"
BEGIN
END_DATA_BLOCK

DATA_BLOCK "Sensor_KR12.3_open"   // DB78
{ S7_Optimized_Access := 'TRUE' }
VERSION : 0.1
// stored: InstanceOfName DI_Single
"DI_Single"
BEGIN
END_DATA_BLOCK

DATA_BLOCK "Sensor_KR12.4_open"   // DB79
{ S7_Optimized_Access := 'TRUE' }
VERSION : 0.1
// stored: InstanceOfName DI_Single
"DI_Single"
BEGIN
END_DATA_BLOCK

DATA_BLOCK "Sensor_KR12.5_open"   // DB80
{ S7_Optimized_Access := 'TRUE' }
VERSION : 0.1
// stored: InstanceOfName DI_Single
"DI_Single"
BEGIN
END_DATA_BLOCK

DATA_BLOCK "Sensor_KR38.5_open"   // DB81
{ S7_Optimized_Access := 'TRUE' }
VERSION : 0.1
// stored: InstanceOfName DI_Single
"DI_Single"
BEGIN
END_DATA_BLOCK

DATA_BLOCK "Sensor_KR38.6_open"   // DB82
{ S7_Optimized_Access := 'TRUE' }
VERSION : 0.1
// stored: InstanceOfName DI_Single
"DI_Single"
BEGIN
END_DATA_BLOCK

DATA_BLOCK "Sensor_water_level_1"   // DB83
{ S7_Optimized_Access := 'TRUE' }
VERSION : 0.1
// stored: InstanceOfName DI_Single
"DI_Single"
BEGIN
END_DATA_BLOCK

DATA_BLOCK "Sensor_water_level_2"   // DB84
{ S7_Optimized_Access := 'TRUE' }
VERSION : 0.1
// stored: InstanceOfName DI_Single
"DI_Single"
BEGIN
END_DATA_BLOCK

DATA_BLOCK "ModbusConnector_DB"   // DB86
{ S7_Optimized_Access := 'TRUE' }
VERSION : 0.1
// stored: InstanceOfName ModbusConnector
"ModbusConnector"
BEGIN
END_DATA_BLOCK

DATA_BLOCK "First_pump_start_DB"   // DB90
{ S7_Optimized_Access := 'TRUE' }
VERSION : 0.1
// stored: InstanceOfName First_pump_start
"First_pump_start"
BEGIN
END_DATA_BLOCK

DATA_BLOCK "State_work_pump_DB"   // DB99
{ S7_Optimized_Access := 'TRUE' }
VERSION : 0.1
// stored: InstanceOfName State_work_pump
"State_work_pump"
BEGIN
END_DATA_BLOCK

// folder: System blocks/Program resources

DATA_BLOCK "Button_UUD_Open_KPPU"   // DB68
{ S7_Optimized_Access := 'TRUE' }
AUTHOR : Simatic
FAMILY : IEC
NAME : IEC_TMR
VERSION : 1.0
// stored: InstanceOfName IEC_TIMER
"IEC_TIMER"
BEGIN
END_DATA_BLOCK

DATA_BLOCK "Cascade_timer"   // DB74
{ S7_Optimized_Access := 'TRUE' }
AUTHOR : Simatic
FAMILY : IEC
NAME : IEC_TMR
VERSION : 1.0
// stored: InstanceOfName IEC_TIMER
"IEC_TIMER"
BEGIN
END_DATA_BLOCK

DATA_BLOCK "UUD_opening_time"   // DB75
{ S7_Optimized_Access := 'TRUE' }
AUTHOR : Simatic
FAMILY : IEC
NAME : IEC_TMR
VERSION : 1.0
// stored: InstanceOfName IEC_TIMER
"IEC_TIMER"
BEGIN
END_DATA_BLOCK

DATA_BLOCK "Timer_cascade_2"   // DB88
{ S7_Optimized_Access := 'TRUE' }
AUTHOR : Simatic
FAMILY : IEC
NAME : IEC_TMR
VERSION : 1.0
// stored: InstanceOfName IEC_TIMER
"IEC_TIMER"
BEGIN
END_DATA_BLOCK

DATA_BLOCK "Timer_Standby_pump"   // DB89
{ S7_Optimized_Access := 'TRUE' }
AUTHOR : Simatic
FAMILY : IEC
NAME : IEC_TMR
VERSION : 1.0
// stored: InstanceOfName IEC_TIMER
"IEC_TIMER"
BEGIN
END_DATA_BLOCK

DATA_BLOCK "Timer_Cascade_3"   // DB91
{ S7_Optimized_Access := 'TRUE' }
AUTHOR : Simatic
FAMILY : IEC
NAME : IEC_TMR
VERSION : 1.0
// stored: InstanceOfName IEC_TIMER
"IEC_TIMER"
BEGIN
END_DATA_BLOCK

DATA_BLOCK "Timer_Cascade_4"   // DB92
{ S7_Optimized_Access := 'TRUE' }
AUTHOR : Simatic
FAMILY : IEC
NAME : IEC_TMR
VERSION : 1.0
// stored: InstanceOfName IEC_TIMER
"IEC_TIMER"
BEGIN
END_DATA_BLOCK

DATA_BLOCK "Timer_Cascade_5"   // DB93
{ S7_Optimized_Access := 'TRUE' }
AUTHOR : Simatic
FAMILY : IEC
NAME : IEC_TMR
VERSION : 1.0
// stored: InstanceOfName IEC_TIMER
"IEC_TIMER"
BEGIN
END_DATA_BLOCK

DATA_BLOCK "UUD1"   // DB94
{ S7_Optimized_Access := 'TRUE' }
AUTHOR : Simatic
FAMILY : IEC
NAME : IEC_TMR
VERSION : 1.0
// stored: InstanceOfName IEC_TIMER
"IEC_TIMER"
BEGIN
END_DATA_BLOCK

// folder: (top level)

FUNCTION_BLOCK "DI_Single"   // FB1, LAD
{ S7_Optimized_Access := 'TRUE' }
VERSION : 0.1
   VAR_INPUT
      input : Bool;
      delay_time : Time;
      filter : Bool;
      reverse : Bool;
   END_VAR
   VAR_OUTPUT
      value : Bool;
   END_VAR
   VAR
      TON : IEC_TIMER;
      TOF : IEC_TIMER;
   END_VAR
   VAR_TEMP   // added for the SCL form of the ladder/FBD networks
      _w1 : Bool;
      _w2 : Bool;
   END_VAR
BEGIN

REGION Network 1
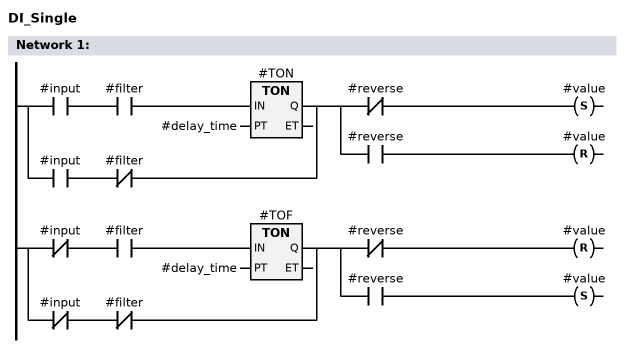
   #TON.TON(IN := #input AND #filter, PT := #delay_time);
   #_w1 := #TON.Q OR (#input AND NOT #filter);
   IF #_w1 AND NOT #reverse THEN #value := TRUE; END_IF;
   IF #_w1 AND #reverse THEN #value := FALSE; END_IF;
   #TOF.TON(IN := NOT #input AND #filter, PT := #delay_time);
   #_w2 := #TOF.Q OR (NOT #input AND NOT #filter);
   IF #_w2 AND NOT #reverse THEN #value := FALSE; END_IF;
   IF #_w2 AND #reverse THEN #value := TRUE; END_IF;
END_REGION
END_FUNCTION_BLOCK

FUNCTION_BLOCK "AI_Sensor"   // FB2, LAD
{ S7_Optimized_Access := 'TRUE' }
VERSION : 0.1
   VAR_INPUT
      In : Int;
      Int_HL : Int := 27468;
      Int_LL : Int := 0;
      Value_HL : Real;
      Value_LL : Real;
   END_VAR
   VAR_OUTPUT
      Value : Real;
      Error : Bool;
   END_VAR
   VAR_TEMP
      In_real : Real;
   END_VAR
BEGIN

REGION Network 1
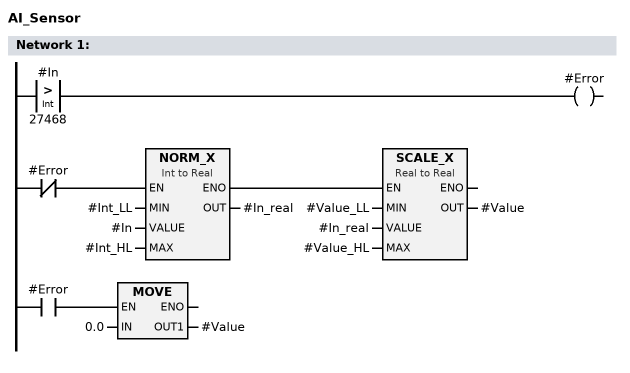
   RUNG wire#powerrail
      { S7_Templates := "SrcType := Int" } GT_Contact(in1 := #In, in2 := 27468)
      Coil( #Error )
   END_RUNG
   RUNG wire#powerrail
      I_Contact( #Error )
      { S7_Templates := "[SrcType := Int, DestType := Real]" } Normalize(min := #Int_LL, value := #In, max := #Int_HL, out => #In_real)
      { S7_Templates := "[SrcType := Real, DestType := Real]" } Scale(min := #Value_LL, value := #In_real, max := #Value_HL, out => #Value)
   END_RUNG
   RUNG wire#powerrail
      Contact( #Error )
      Move(in := 0.0, out1 => #Value)
   END_RUNG
   // the same network as SCL:
   #Error := #In > 27468;
   IF NOT #Error THEN
       #In_real := NORM_X(MIN := #Int_LL, VALUE := #In, MAX := #Int_HL);
       #Value := SCALE_X(MIN := #Value_LL, VALUE := #In_real, MAX := #Value_HL);
   END_IF;
   IF #Error THEN #Value := 0.0; END_IF;
END_REGION
END_FUNCTION_BLOCK

FUNCTION_BLOCK "AI_Redundancy"   // FB3, SCL
{ S7_Optimized_Access := 'TRUE' }
VERSION : 0.1
   VAR_INPUT
      IN_AI_01 : Real;   // Сигнал 01
      IN_AI_02 : Real;   // Сигнал 02
      IN_Err_Proc : Real;   // Предельная разность сигналов
   END_VAR
   VAR_OUTPUT
      OUT_Error : Bool;   // Сигналы различаются больше чем на IN_Err_Proc %
      OUT_Result : Real;   // Результатирующий сигнал
   END_VAR
   VAR
      Error_1 : Real;
      Error_2 : Real;
   END_VAR
BEGIN
   #Error_1 := ABS(#IN_AI_01 - #IN_AI_02)*100.0 / #IN_AI_02;
   #Error_2 := ABS(#IN_AI_01 - #IN_AI_02)*100.0/ #IN_AI_01;
   IF #Error_1 > #IN_Err_Proc OR #Error_2 > #IN_Err_Proc THEN
       #OUT_Error := TRUE;
   ELSE
       #OUT_Error := FALSE;
   END_IF;

   IF #OUT_Error THEN
       #OUT_Result := MAX(IN1 := #IN_AI_01, IN2 := #IN_AI_02);
   ELSE
       #OUT_Result := (#IN_AI_01 + #IN_AI_02) / 2;
   END_IF;
END_FUNCTION_BLOCK

FUNCTION_BLOCK "Standby_Pump/Compressor_Error"   // FB4, LAD
{ S7_Optimized_Access := 'TRUE' }
VERSION : 0.1
   VAR_INPUT
      DQ : Bool;
      STATE_Switch : Bool;
      STATE_Starter : Bool;
   END_VAR
   VAR_OUTPUT
      Error : Bool;
   END_VAR
   VAR
      TP : IEC_TIMER;
      TON : IEC_TIMER;
   END_VAR
BEGIN

REGION Network 1
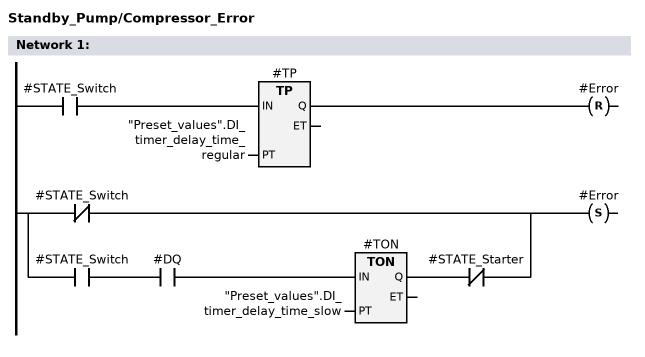
   #TP.TP(IN := #STATE_Switch, PT := "Preset_values".DI_timer_delay_time_regular);
   IF #TP.Q THEN #Error := FALSE; END_IF;
   #TON.TON(IN := #STATE_Switch AND #DQ, PT := "Preset_values".DI_timer_delay_time_slow);
   IF NOT #STATE_Switch OR (#TON.Q AND NOT #STATE_Starter) THEN #Error := TRUE; END_IF;
END_REGION
END_FUNCTION_BLOCK

FUNCTION_BLOCK "Pump_Error"   // FB5, LAD
{ S7_Optimized_Access := 'TRUE' }
VERSION : 0.1
   VAR_INPUT
      DQ : Bool;
      STATE_Switch : Bool;
      STATE_Starter : Bool;
      SENSOR_Ball_Valve : Bool;
      SENSOR_High_Pressure_Pump : Real;
      SENSOR_High_Pressure_Pump_Error : Bool;
   END_VAR
   VAR_OUTPUT
      Error : Bool;
   END_VAR
   VAR
      TP : IEC_TIMER;
      TON_1 : IEC_TIMER;
      TON_2 : IEC_TIMER;
      Error_1 : Bool;
      Error_2 : Bool;
   END_VAR
BEGIN

REGION Network 1
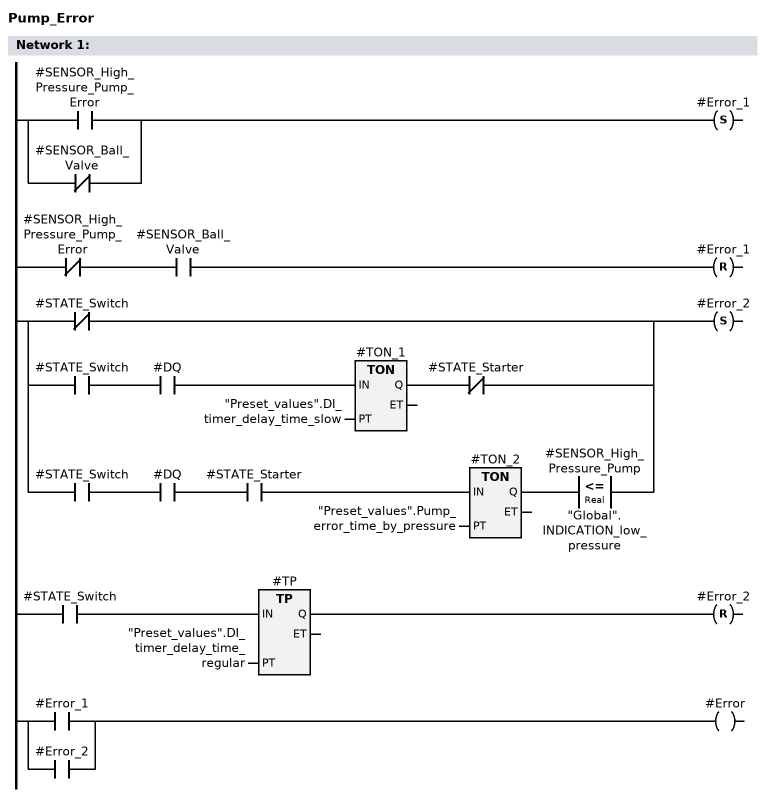
   IF #SENSOR_High_Pressure_Pump_Error OR NOT #SENSOR_Ball_Valve THEN #Error_1 := TRUE; END_IF;
   IF NOT #SENSOR_High_Pressure_Pump_Error AND #SENSOR_Ball_Valve THEN #Error_1 := FALSE; END_IF;
   #TON_1.TON(IN := #STATE_Switch AND #DQ, PT := "Preset_values".DI_timer_delay_time_slow);
   #TON_2.TON(IN := #STATE_Switch AND #DQ AND #STATE_Starter, PT := "Preset_values".Pump_error_time_by_pressure);
   IF NOT #STATE_Switch OR (#TON_1.Q AND NOT #STATE_Starter) OR (#TON_2.Q AND (#SENSOR_High_Pressure_Pump <= "Global".INDICATION_low_pressure)) THEN
       #Error_2 := TRUE;
   END_IF;
   #TP.TP(IN := #STATE_Switch, PT := "Preset_values".DI_timer_delay_time_regular);
   IF #TP.Q THEN #Error_2 := FALSE; END_IF;
   #Error := #Error_1 OR #Error_2;
END_REGION
END_FUNCTION_BLOCK

FUNCTION_BLOCK "First_pump_start"   // FB6, SCL
{ S7_Optimized_Access := 'TRUE' }
VERSION : 0.1
   VAR_INPUT
      Total_pumps : Int;
   END_VAR
   VAR_IN_OUT
      Control_pump_1 : Bool;
      Control_pump_2 : Bool := false;
      Control_pump_3 : Bool := false;
      Control_pump_4 : Bool := false;
      Control_pump_5 : Bool := false;
   END_VAR
   VAR_TEMP
      "Counter" : Int;
      Start_pump : Int;
   END_VAR
BEGIN
   IF NOT "Global".BUTTON_Global_Stop
       AND NOT "MB_BUTTON_GLOBAL_STOP"
       AND "Global".MODE_auto
       AND NOT "Global".MODE_standby
       AND NOT "Global".ERROR_global
       AND "Global".SIGNAL_fire
       AND NOT "Global".SIGNAL_first_pump_has_started
   THEN
       FOR #Counter := 1 TO #Total_pumps DO
           IF NOT "Pumps_data".Error_pump[#Counter]
               AND NOT "Pumps_data".State_work_pump[#Counter]
           THEN
               CASE #Counter OF
                   1:  
                       #Control_pump_1 := true;
                       ;
                   2:  
                       #Control_pump_2 := true;
                       ;
                   3:  
                       #Control_pump_3 := true;
                       ;
                   4:  
                       #Control_pump_4 := true;
                       ;
                   5:  
                       #Control_pump_5 := true;
                       ;
               END_CASE;
               "Global".SIGNAL_first_pump_has_started := TRUE;
               EXIT;
           END_IF;
       END_FOR;
   END_IF;
END_FUNCTION_BLOCK

FUNCTION_BLOCK "State_work_pump"   // FB7, SCL
{ S7_Optimized_Access := 'TRUE' }
VERSION : 0.1
   VAR_INPUT
      Total_pumps : Int;
   END_VAR
   VAR_TEMP
      "Counter" : Int;
   END_VAR
BEGIN
   FOR #Counter := 1 TO #Total_pumps DO
       IF "Pumps_data".State_starter_pump[#Counter] AND "Pumps_data".State_switch_pump[#Counter] THEN
           "Pumps_data".State_work_pump[#Counter] := true;
       ELSE
           "Pumps_data".State_work_pump[#Counter] := FALSE;
       END_IF;
   END_FOR;
END_FUNCTION_BLOCK

FUNCTION_BLOCK "Button_open UUD"   // FB8, SCL
{ S7_Optimized_Access := 'TRUE' }
VERSION : 0.1
   VAR_INPUT
      button : Bool;
      pressure : Real;
      error : Bool;
      aps : Bool;
   END_VAR
   VAR_OUTPUT
      output : Bool;
      signal_opened : Bool;
   END_VAR
   VAR
      "Time" : Time := T#1s;
      start : Bool;
   END_VAR
   VAR_TEMP
      Count : Int;
   END_VAR
BEGIN
   IF #button OR #aps AND NOT #error THEN
       #Count := 1;
       #start := true;
       IF #Count = 1 THEN
           #output := TRUE;
           "UUD_opening_time".TON(IN := #start,
                                  PT := #Time);
           IF #pressure < 5 THEN
               #Count := 2;
               #output := FALSE;
           ELSE
               #Count := 0;
               #output := FALSE;
               #signal_opened := TRUE;
           END_IF;
       END_IF;

       IF #Count = 2 THEN
           #output := TRUE;
           "UUD_opening_time".TON(IN := #start,
                                  PT := #Time);
           IF #pressure < 5 THEN
               #Count := 3;
               #output := FALSE;
           ELSE
               #Count := 0;
               #output := FALSE;
               #signal_opened := TRUE;
           END_IF;
       END_IF;

       IF #Count = 3 THEN
           #output := TRUE;
           "UUD_opening_time".TON(IN := #start,
                                  PT := #Time);
           IF #pressure < 5 THEN
               #Count := 0;
               #output := FALSE;
           ELSE
               #Count := 0;
               #output := FALSE;
               #signal_opened := TRUE;
           END_IF;

       END_IF;
   END_IF;
END_FUNCTION_BLOCK

FUNCTION_BLOCK "Sound_PTO"   // FB10, LAD
{ S7_Optimized_Access := 'TRUE' }
VERSION : 0.1
   VAR_INPUT
      Hardware_ID : Hw_Pto;
      Button_sound_off : Bool;
      ERROR_any : Bool;
      SIGNAL_fire : Bool;
      STATE_work_any_pump : Bool;
      Error_frequency : UDInt := 1;
      Fire_frequency : UDInt := 2;
      Work_frequency : UDInt := 50;
   END_VAR
   VAR_OUTPUT
      Led_sound_off : Bool;
   END_VAR
   VAR
      Frequency : UDInt;
      Sound_off : Bool;
   END_VAR
   VAR_TEMP   // added for the SCL form of the ladder/FBD networks
      _w1 : Bool;
      _w2 : Bool;
   END_VAR
BEGIN

REGION Network 1
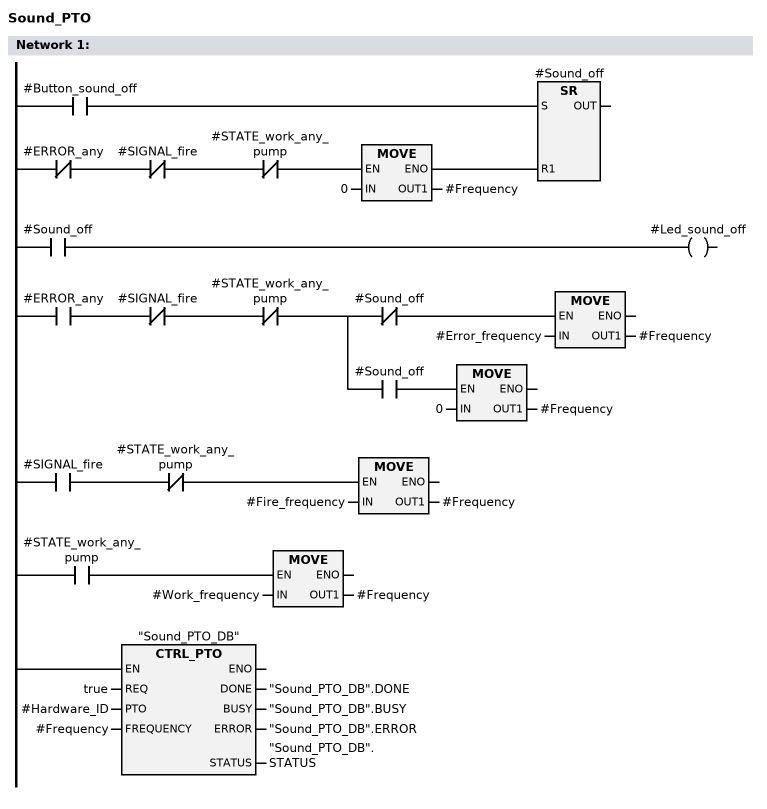
   #_w1 := NOT #ERROR_any AND NOT #SIGNAL_fire AND NOT #STATE_work_any_pump;
   IF #_w1 THEN #Frequency := 0; END_IF;
   IF #Button_sound_off THEN
       #Sound_off := TRUE;   // SR flip-flop
   END_IF;
   IF #_w1 THEN #Sound_off := FALSE; END_IF;
   #Led_sound_off := #Sound_off;
   #_w2 := #ERROR_any AND NOT #SIGNAL_fire AND NOT #STATE_work_any_pump;
   IF #_w2 AND NOT #Sound_off THEN #Frequency := #Error_frequency; END_IF;
   IF #_w2 AND #Sound_off THEN #Frequency := 0; END_IF;
   IF #SIGNAL_fire AND NOT #STATE_work_any_pump THEN #Frequency := #Fire_frequency; END_IF;
   IF #STATE_work_any_pump THEN #Frequency := #Work_frequency; END_IF;
   "Sound_PTO_DB"(REQ := true,   // CTRL_PTO
                  PTO := #Hardware_ID,
                  FREQUENCY := #Frequency,
                  DONE => "Sound_PTO_DB".DONE,
                  BUSY => "Sound_PTO_DB".BUSY,
                  ERROR => "Sound_PTO_DB".ERROR,
                  STATUS => "Sound_PTO_DB".STATUS);
END_REGION
END_FUNCTION_BLOCK

FUNCTION_BLOCK "Data_push_to_HMI"   // FB12, SCL
{ S7_Optimized_Access := 'TRUE' }
VERSION : 0.1
BEGIN
   "HMI_MODE_AUTO" := "Global".MODE_auto;
   "HMI_MODE_MANUAL" := "Global".MODE_manual;
   "HMI_MODE_BLOCKED" := "Global".MODE_blocked;
   "HMI_MODE_STANDBY" := "Global".MODE_standby;
   "HMI_ERROR_ANY" := "Global".ERROR_any;
   "HMI_ERROR_INLET_PRESSURE_LOW" := "Global".ERROR_inlet_pressure_low;
   "HMI_ERROR_PUMP1" := "Pumps_data".Error_pump[1];
   "HMI_ERROR_PUMP2" := "Pumps_data".Error_pump[2];
   "HMI_ERROR_PUMP3" := "Pumps_data".Error_pump[3];
   "HMI_ERROR_PUMP4" := "Pumps_data".Error_pump[4];
   "HMI_ERROR_PUMP5" := "Pumps_data".Error_pump[5];
   "HMI_ERROR_PRESSURE_SENSOR_PUMP1" := "Pumps_data".Pump_sensor_error[1];
   "HMI_ERROR_PRESSURE_SENSOR_PUMP2" := "Pumps_data".Pump_sensor_error[2];
   "HMI_ERROR_PRESSURE_SENSOR_PUMP3" := "Pumps_data".Pump_sensor_error[3];
   "HMI_ERROR_PRESSURE_SENSOR_PUMP4" := "Pumps_data".Pump_sensor_error[4];
   "HMI_ERROR_PRESSURE_SENSOR_PUMP5" := "Pumps_data".Pump_sensor_error[5];
   "HMI_BUTTON_GLOBAL_STOP" := "Global".BUTTON_Global_Stop;
   "HMI_ERROR_STANDBY_PUMP" := "Pumps_data".Error_standby_pump;
   "HMI_SENSOR_FLOW_UUS1" := "Section_valves_data".SENSOR_flow_UUS[1];
   "HMI_SENSOR_FLOW_UUS2" := "Section_valves_data".SENSOR_flow_UUS[2];
   "HMI_SENSOR_FLOW_UUS3" := "Section_valves_data".SENSOR_flow_UUS[3];
   "HMI_SENSOR_FLOW_UUS4" := "Section_valves_data".SENSOR_flow_UUS[4];
   "HMI_SENSOR_FLOW_UUS5" := "Section_valves_data".SENSOR_flow_UUS[5];
   "HMI_SIGNAL_OPEN_UUS1" := "Section_valves_data".SENSOR_open_UUS[1];
   "HMI_SIGNAL_OPEN_UUS2" := "Section_valves_data".SENSOR_open_UUS[2];
   "HMI_SIGNAL_OPEN_UUS3" := "Section_valves_data".SENSOR_open_UUS[3];
   "HMI_SIGNAL_OPEN_UUS4" := "Section_valves_data".SENSOR_open_UUS[4];
   "HMI_SIGNAL_OPEN_UUS5" := "Section_valves_data".SENSOR_open_UUS[5];
   "HMI_SENSOR_ERROR_UUS1" := "Section_valves_data".SENSOR_ERROR_UUS[1];
   "HMI_SENSOR_ERROR_UUS2" := "Section_valves_data".SENSOR_ERROR_UUS[2];
   "HMI_SENSOR_ERROR_UUS3" := "Section_valves_data".SENSOR_ERROR_UUS[3];
   "HMI_SENSOR_ERROR_UUS4" := "Section_valves_data".SENSOR_ERROR_UUS[4];
   "HMI_SENSOR_ERROR_UUS5" := "Section_valves_data".SENSOR_ERROR_UUS[5];
   "HMI_SENSOR_OPEN_KP38.1" := "Ball_valves_data".SENSOR_KR38_open[1];
   "HMI_SENSOR_OPEN_KP38.2" := "Ball_valves_data".SENSOR_KR38_open[2];
   "HMI_SENSOR_OPEN_KP38.3" := "Ball_valves_data".SENSOR_KR38_open[3];
   "HMI_SENSOR_OPEN_KP38.4" := "Ball_valves_data".SENSOR_KR38_open[4];
   "HMI_SENSOR_OPEN_KP38.5" := "Ball_valves_data".SENSOR_KR38_open[5];
   "HMI_SENSOR_OPEN_KP38.6" := "Ball_valves_data".SENSOR_KR38_open[6];
   "HMI_STATE_380_MAIN" := "Global".STATE_380_main;
   "HMI_STATE_380_BACKUP" := "Global".STATE_380_backup;
   "HMI_STATE_220_INNER" := "Global".STATE_220_inner;
   "HMI_STATE_220_OUTER" := "Global".STATE_220_outer;
   "HMI_STATE_DOOR_OPENED" := "Global".STATE_door_opened;
   "HMI_ERROR_UNDERWATER" := "Global".ERROR_underwater;
   "HMI_ERROR_NO_WATER" := "Global".ERROR_no_water;
   "HMI_ERROR_NO_WATER_FIRE" := "Global".ERROR_no_water_fire;
   "HMI_ERROR_GLOBAL" := "Global".ERROR_global;
   "HMI_ERROR_UUS" := "Global".ERROR_UUS;
   "HMI_ERROR_UUS_ANY" := "Global".ERROR_UUS_any;
   "HMI_ERROR_PUMPS" := "Global".ERROR_PUMPS;
   "HMI_ERROR_BALL_VALVE_ANY" := "Global".ERROR_ball_valve_any;
   "HMI_SIGNAL_FIRE" := "Global".SIGNAL_fire;
   "HMI_SENSOR_PRESSURE_PUMP1" := "Global".SENSOR_high_pressure_pump_1;
   "HMI_SENSOR_PRESSURE_PUMP2" := "Global".SENSOR_high_pressure_pump_2;
   "HMI_SENSOR_PRESSURE_PUMP3" := "Global".SENSOR_high_pressure_pump_3;
   "HMI_SENSOR_PRESSURE_PUMP4" := "Global".SENSOR_high_pressure_pump_4;
   "HMI_SENSOR_PRESSURE_PUMP5" := "Global".SENSOR_high_pressure_pump_5;
   "HMI_SENSOR_INDICATION_PRESSURE_LOW" := "Global".INDICATION_low_pressure;
   "HMI_SENSOR_INDICATION_PRESSURE_HIGH" := "Global".INDICATION_high_pressure;
   "HMI_STATE_WORK_PUMP1" := "Pumps_data".State_work_pump[1];
   "HMI_STATE_WORK_PUMP2" := "Pumps_data".State_work_pump[2];
   "HMI_STATE_WORK_PUMP3" := "Pumps_data".State_work_pump[3];
   "HMI_STATE_WORK_PUMP4" := "Pumps_data".State_work_pump[4];
   "HMI_STATE_WORK_PUMP5" := "Pumps_data".State_work_pump[5];
   "HMI_STATE_WORK_STANDBY_PUMP" := "Pumps_data".State_work_standby_pump;
   "HMI_STATE_WORK_ANY_PUMP" := "Pumps_data".State_work_any_pump;
   "HMI_WATER_LEVEL_FULL" := "Water_control".Water_level_full;
   "HMI_SIGNAL_NEED_REPLENISH_1" := "Water_control".Signal_need_replenish_1;
   "HMI_SIGNAL_NEED_REPLENISH_2" := "Water_control".Signal_need_replenish_2;
   "HMI_ERROR_UUD1" := "Section_valves_data".SENSOR_ERROR_UUD1;
   "HMI_ERROR_DRAIN_PUMP" := "Pumps_data".Error_drain_pump;
   "HMI_STATE_WORK_DRAIN_PUMP" := "Pumps_data".State_work_drain_pump;
   "HMI_Sensor_water_level_1" := "Global".Sensor_water_level_1;
   "HMI_Sensor_water_level_2" := "Global".Sensor_water_level_2;
   "HMI_Sensor_water_level_3" := "Global".Sensor_water_level_3;
   "HMI_Sensor_drain_work" := "Global".Sensor_drain_work;
   "HMI_Sensor_drain_overflow" := "Global".Sensor_drain_overflow;
   "HMI_SENSOR_OPEN_KP12.1" := "Ball_valves_data".SENSOR_KR12_open[1];
   "HMI_SENSOR_OPEN_KP12.2" := "Ball_valves_data".SENSOR_KR12_open[2];
   "HMI_SENSOR_OPEN_KP12.3" := "Ball_valves_data".SENSOR_KR12_open[3];
   "HMI_SENSOR_OPEN_KP12.4" := "Ball_valves_data".SENSOR_KR12_open[4];
   "HMI_SENSOR_OPEN_KP12.5" := "Ball_valves_data".SENSOR_KR12_open[5];
END_FUNCTION_BLOCK

FUNCTION_BLOCK "Data_push_to_MODBUS"   // FB13, SCL
{ S7_Optimized_Access := 'TRUE' }
VERSION : 0.1
BEGIN
   "MB_MODE_AUTO" := "Global".MODE_auto;
   "MB_MODE_MANUAL" := "Global".MODE_manual;
   "MB_MODE_BLOCKED" := "Global".MODE_blocked;
   "MB_MODE_STANDBY" := "Global".MODE_standby;
   "MB_ERROR_ANY" := "Global".ERROR_any;
   "MB_ERROR_INLET_PRESSURE_LOW" := "Global".ERROR_inlet_pressure_low;
   "MB_ERROR_PUMP1" := "Pumps_data".Error_pump[1];
   "MB_ERROR_PUMP2" := "Pumps_data".Error_pump[2];
   "MB_ERROR_PUMP3" := "Pumps_data".Error_pump[3];
   "MB_ERROR_PUMP4" := "Pumps_data".Error_pump[4];
   "MB_ERROR_PUMP5" := "Pumps_data".Error_pump[5];
   "MB_ERROR_PRESSURE_SENSOR_PUMP1" := "Pumps_data".Pump_sensor_error[1];
   "MB_ERROR_PRESSURE_SENSOR_PUMP2" := "Pumps_data".Pump_sensor_error[2];
   "MB_ERROR_PRESSURE_SENSOR_PUMP3" := "Pumps_data".Pump_sensor_error[3];
   "MB_ERROR_PRESSURE_SENSOR_PUMP4" := "Pumps_data".Pump_sensor_error[4];
   "MB_ERROR_PRESSURE_SENSOR_PUMP5" := "Pumps_data".Pump_sensor_error[5];
   "MB_BUTTON_GLOBAL_STOP" := "Global".BUTTON_Global_Stop;
   "MB_ERROR_STANDBY_PUMP" := "Pumps_data".Error_standby_pump;
   "MB_SENSOR_FLOW_UUS1" := "Section_valves_data".SENSOR_flow_UUS[1];
   "MB_SENSOR_FLOW_UUS2" := "Section_valves_data".SENSOR_flow_UUS[2];
   "MB_SENSOR_FLOW_UUS3" := "Section_valves_data".SENSOR_flow_UUS[3];
   "MB_SENSOR_FLOW_UUS4" := "Section_valves_data".SENSOR_flow_UUS[4];
   "MB_SENSOR_FLOW_UUS5" := "Section_valves_data".SENSOR_flow_UUS[5];
   "MB_SIGNAL_OPEN_UUS1" := "Section_valves_data".SENSOR_open_UUS[1];
   "MB_SIGNAL_OPEN_UUS2" := "Section_valves_data".SENSOR_open_UUS[2];
   "MB_SIGNAL_OPEN_UUS3" := "Section_valves_data".SENSOR_open_UUS[3];
   "MB_SIGNAL_OPEN_UUS4" := "Section_valves_data".SENSOR_open_UUS[4];
   "MB_SIGNAL_OPEN_UUS5" := "Section_valves_data".SENSOR_open_UUS[5];
   "MB_SENSOR_ERROR_UUS1" := "Section_valves_data".SENSOR_ERROR_UUS[1];
   "MB_SENSOR_ERROR_UUS2" := "Section_valves_data".SENSOR_ERROR_UUS[2];
   "MB_SENSOR_ERROR_UUS3" := "Section_valves_data".SENSOR_ERROR_UUS[3];
   "MB_SENSOR_ERROR_UUS4" := "Section_valves_data".SENSOR_ERROR_UUS[4];
   "MB_SENSOR_ERROR_UUS5" := "Section_valves_data".SENSOR_ERROR_UUS[5];
   "MB_SENSOR_OPEN_KP38.1" :="Ball_valves_data".SENSOR_KR38_open[1];
   "MB_SENSOR_OPEN_KP38.2" :="Ball_valves_data".SENSOR_KR38_open[2];
   "MB_SENSOR_OPEN_KP38.3" :="Ball_valves_data".SENSOR_KR38_open[3];
   "MB_SENSOR_OPEN_KP38.4" :="Ball_valves_data".SENSOR_KR38_open[4];
   "MB_SENSOR_OPEN_KP38.5" :="Ball_valves_data".SENSOR_KR38_open[5];
   "MB_SENSOR_OPEN_KP38.6" :="Ball_valves_data".SENSOR_KR38_open[6];
   "MB_STATE_380_MAIN" := "Global".STATE_380_main;
   "MB_STATE_380_BACKUP" := "Global".STATE_380_backup;
   "MB_STATE_220_INNER" := "Global".STATE_220_inner;
   "MB_STATE_220_OUTER" := "Global".STATE_220_outer;
   "MB_STATE_DOOR_OPENED" := "Global".STATE_door_opened;
   "MB_ERROR_UNDERWATER" := "Global".ERROR_underwater;
   "MB_ERROR_NO_WATER" := "Global".ERROR_no_water;
   "MB_ERROR_NO_WATER_FIRE" := "Global".ERROR_no_water_fire;
   "MB_ERROR_GLOBAL" := "Global".ERROR_global;
   "MB_ERROR_UUS" := "Global".ERROR_UUS;
   "MB_ERROR_UUS_ANY" := "Global".ERROR_UUS_any;
   "MB_ERROR_PUMPS" := "Global".ERROR_PUMPS;
   "MB_ERROR_BALL_VALVE_ANY" := "Global".ERROR_ball_valve_any;
   "MB_SIGNAL_FIRE" := "Global".SIGNAL_fire;
   "MB_SENSOR_PRESSURE_PUMP1" := "Global".SENSOR_high_pressure_pump_1;
   "MB_SENSOR_PRESSURE_PUMP2" := "Global".SENSOR_high_pressure_pump_2;
   "MB_SENSOR_PRESSURE_PUMP3" := "Global".SENSOR_high_pressure_pump_3;
   "MB_SENSOR_PRESSURE_PUMP4" := "Global".SENSOR_high_pressure_pump_4;
   "MB_SENSOR_PRESSURE_PUMP5" := "Global".SENSOR_high_pressure_pump_5;
   "MB_SENSOR_INDICATION_PRESSURE_LOW" := "Global".INDICATION_low_pressure;
   "MB_SENSOR_INDICATION_PRESSURE_HIGH" := "Global".INDICATION_high_pressure;
   "MB_STATE_WORK_PUMP1" := "Pumps_data".State_work_pump[1];
   "MB_STATE_WORK_PUMP2" := "Pumps_data".State_work_pump[2];
   "MB_STATE_WORK_PUMP3" := "Pumps_data".State_work_pump[3];
   "MB_STATE_WORK_PUMP4" := "Pumps_data".State_work_pump[4];
   "MB_STATE_WORK_PUMP5" := "Pumps_data".State_work_pump[5];
   "MB_STATE_WORK_STANDBY_PUMP" := "Pumps_data".State_work_standby_pump;
   "MB_STATE_WORK_ANY_PUMP" := "Pumps_data".State_work_any_pump;
   "MB_WATER_LEVEL_FULL" := "Water_control".Water_level_full;
   "MB_SIGNAL_NEED_REPLENISH_1" := "Water_control".Signal_need_replenish_1;
   "MB_SIGNAL_NEED_REPLENISH_2" := "Water_control".Signal_need_replenish_2;
   "MB_ERROR_UUD1" := "Section_valves_data".SENSOR_ERROR_UUD1;
   "MB_ERROR_DRAIN_PUMP" := "Pumps_data".Error_drain_pump;
   "MB_STATE_WORK_DRAIN_PUMP" := "Pumps_data".State_work_drain_pump;
   "MB_Sensor_water_level_1" := "Global".Sensor_water_level_1;
   "MB_Sensor_water_level_2" := "Global".Sensor_water_level_2;
   "MB_Sensor_water_level_3" := "Global".Sensor_water_level_3;
   "MB_Sensor_drain_work" := "Global".Sensor_drain_work;
   "MB_Sensor_drain_overflow" := "Global".Sensor_drain_overflow;
   "MB_SENSOR_OPEN_KP12.1" :="Ball_valves_data".SENSOR_KR12_open[1];
   "MB_SENSOR_OPEN_KP12.2" :="Ball_valves_data".SENSOR_KR12_open[2];
   "MB_SENSOR_OPEN_KP12.3" :="Ball_valves_data".SENSOR_KR12_open[3];
   "MB_SENSOR_OPEN_KP12.4" :="Ball_valves_data".SENSOR_KR12_open[4];
   "MB_SENSOR_OPEN_KP12.5" :="Ball_valves_data".SENSOR_KR12_open[5];
END_FUNCTION_BLOCK

FUNCTION_BLOCK "Cascade_start_stop"   // FB14, SCL
{ S7_Optimized_Access := 'TRUE' }
VERSION : 0.1
   VAR_INPUT
      Total_pumps : Int;
   END_VAR
   VAR_IN_OUT
      Pump1 : Bool;
      Pump2 : Bool;
      Pump3 : Bool;
      Pump4 : Bool;
      Pump5 : Bool;
   END_VAR
   VAR_TEMP
      "Counter" : Int;
      Start_cascade_pump : Int;
      "Timer" : Bool;
      Stop_cascade_pump : Int;
      Command : String;
   END_VAR
BEGIN
   IF NOT "Global".BUTTON_Global_Stop
       AND NOT "MB_BUTTON_GLOBAL_STOP"
       AND "Global".MODE_auto
       AND NOT "Global".MODE_standby
       AND NOT "Global".ERROR_global
       AND "Global".SIGNAL_fire
       AND "Global".SIGNAL_first_pump_has_started
   THEN
       FOR #Counter := #Total_pumps TO 1 DO
           IF NOT "Pumps_data".Error_pump[#Counter]
               AND "Pumps_data".State_work_pump[#Counter]
               AND "Global".INDICATION_high_pressure <= "Preset_values".Pressure_cascade_start
               AND #Counter < #Total_pumps
           THEN
               #Start_cascade_pump := #Counter + 1;
               #Command := 'Start';
           END_IF;
           IF NOT "Pumps_data".Error_pump[#Counter]
               AND "Pumps_data".State_work_pump[#Counter]
               AND "Global".INDICATION_high_pressure >= "Preset_values".Pressure_cascade_stop
           THEN
               #Stop_cascade_pump := #Counter;
               #Command := 'Stop';
           END_IF;
       END_FOR;

       CASE #Counter OF
           5:
               #Timer := FALSE;
               IF #Command = 'Start' THEN
                   ;
               ELSIF #Command = 'Stop' THEN
                   #Pump5 := FALSE;
               END_IF;
           4:
               #Timer := TRUE;
               IF #Command = 'Start' THEN
                   "Cascade_timer".TON(IN := #Timer,
                                       PT := "Preset_values".Timer_cascade_start);
                   #Pump5 := TRUE;
               ELSIF #Command = 'Stop' THEN
                   #Pump4 := FALSE;
               END_IF;
           3:
               #Timer := TRUE;
               IF #Command = 'Start' THEN
                   "Cascade_timer".TON(IN := #Timer,
                                       PT := "Preset_values".Timer_cascade_start);
                   #Pump4 := TRUE;
               ELSIF #Command = 'Stop' THEN
                   #Pump3 := FALSE;
               END_IF;
           2:
               #Timer := TRUE;
               IF #Command = 'Start' THEN
                   "Cascade_timer".TON(IN := #Timer,
                                       PT := "Preset_values".Timer_cascade_start);
                   #Pump3 := TRUE;
               ELSIF #Command = 'Stop' THEN
                   #Pump2 := FALSE;
               END_IF;
           1:
               #Timer := TRUE;
               IF #Command = 'Start' THEN
                   "Cascade_timer".TON(IN := #Timer,
                                       PT := "Preset_values".Timer_cascade_start);
                   #Pump2 := TRUE;
               ELSIF #Command = 'Stop' THEN
                   IF NOT #Pump1 THEN
                       #Pump1 := TRUE;
                       ;
                   END_IF;


               END_IF;

       END_CASE;

       ;
   END_IF;
END_FUNCTION_BLOCK

FUNCTION_BLOCK "ModbusConnector"   // FB15, SCL
{ S7_Optimized_Access := 'TRUE' }
VERSION : 0.1
   VAR
      instModbusCommLoad : Modbus_Comm_Load;
      instModbusMaster : Modbus_Master;
      Init : Bool := TRUE;
      PORT : Port := 269;
      BAUD : UDInt := 9600;
      STOP_BITS : USInt := 1;
      PARITY : UInt := 0;
      Read_REGS : Word;
      "Step" : UInt;
      Write_REGS : Array[0..38] of Word;
   END_VAR
BEGIN
   IF #Init THEN
       #Step := 2;
       #instModbusCommLoad.MODE := 4;
       #instModbusCommLoad.STOP_BITS := #STOP_BITS;
   END_IF;

   #instModbusCommLoad(REQ := #Init,
                       "PORT" := #PORT,
                       BAUD := #BAUD,
                       PARITY := #PARITY,
                       MB_DB := #instModbusMaster.MB_DB);

   #Init := FALSE;

   CASE #Step OF
   1:

   #instModbusMaster(REQ := TRUE,
                     MB_ADDR := 1,
                     MODE := 0,
                     DATA_ADDR := 40001,
                     DATA_LEN := 1,
                     DATA_PTR := #Read_REGS);
   IF #instModbusMaster.DONE THEN
       #Step := 2;
       "ReadHolding" := #Read_REGS;

       #Write_REGS[0] := "WriteHoldingRegister_00";
       #Write_REGS[1] := "WriteHoldingRegister_01";
       #Write_REGS[2] := "WriteHoldingRegister_02";
       #Write_REGS[3] := "WriteHoldingRegister_03";
       #Write_REGS[4] := "WriteHoldingRegister_04";
       #Write_REGS[5] := "WriteHoldingRegister_05";
       #Write_REGS[6] := "WriteHoldingRegister_06";
       #Write_REGS[7] := "WriteHoldingRegister_07";
       #Write_REGS[8] := "WriteHoldingRegister_08";
       #Write_REGS[9] := "WriteHoldingRegister_09";
       #Write_REGS[10] := "WriteHoldingRegister_10";
       #Write_REGS[11] := "WriteHoldingRegister_11";
       #Write_REGS[12] := "WriteHoldingRegister_12";
       #Write_REGS[13] := "WriteHoldingRegister_13";
       #Write_REGS[14] := "WriteHoldingRegister_14";
       #Write_REGS[15] := "WriteHoldingRegister_15";
       #Write_REGS[16] := "WriteHoldingRegister_16";
       #Write_REGS[17] := "WriteHoldingRegister_17";
       #Write_REGS[18] := "WriteHoldingRegister_18";
       #Write_REGS[19] := "WriteHoldingRegister_19";
       #Write_REGS[20] := "WriteHoldingRegister_20";
       #Write_REGS[21] := "WriteHoldingRegister_21";
       #Write_REGS[22] := "WriteHoldingRegister_22";
       #Write_REGS[23] := "WriteHoldingRegister_23";
       #Write_REGS[24] := "WriteHoldingRegister_24";
       #Write_REGS[25] := "WriteHoldingRegister_25";
       #Write_REGS[26] := "WriteHoldingRegister_26";
       #Write_REGS[27] := "WriteHoldingRegister_27";
       #Write_REGS[28] := "WriteHoldingRegister_28";
       #Write_REGS[29] := "WriteHoldingRegister_29";
       #Write_REGS[30] := "WriteHoldingRegister_30";
       #Write_REGS[31] := "WriteHoldingRegister_31";
       #Write_REGS[32] := "WriteHoldingRegister_32";
       #Write_REGS[33] := "WriteHoldingRegister_33";
       #Write_REGS[34] := "WriteHoldingRegister_34";
       #Write_REGS[35] := "WriteHoldingRegister_35";
       #Write_REGS[36] := "WriteHoldingRegister_36";
       #Write_REGS[37] := "WriteHoldingRegister_37";
       #Write_REGS[38] := "WriteHoldingRegister_38";


   END_IF;
   IF #instModbusMaster.ERROR THEN
       #Step := 2;
   END_IF;
   2:
       #instModbusMaster(REQ := TRUE,
                         MB_ADDR := 1,
                         MODE := 1,
                         DATA_ADDR := 40002,
                         DATA_LEN := 39,
                         DATA_PTR := #Write_REGS);
       IF #instModbusMaster.DONE THEN
           #Step := 1;


       END_IF;
       IF #instModbusMaster.ERROR THEN
           #Step := 1;
       END_IF;
   END_CASE;
END_FUNCTION_BLOCK

FUNCTION "DI_All" : Void   // FC1, LAD
{ S7_Optimized_Access := 'TRUE' }
VERSION : 0.1
   VAR_TEMP   // added for the SCL form of the ladder/FBD networks
      _w1 : Bool;
      _w2 : Bool;
      _w3 : Bool;
      _w4 : Bool;
      _w5 : Bool;
      _w6 : Bool;
      _w7 : Bool;
      _w8 : Bool;
      _w9 : Bool;
      _w10 : Bool;
      _w11 : Bool;
      _w12 : Bool;
   END_VAR
BEGIN

REGION Network 1: Дискретные входы состояния шкафа
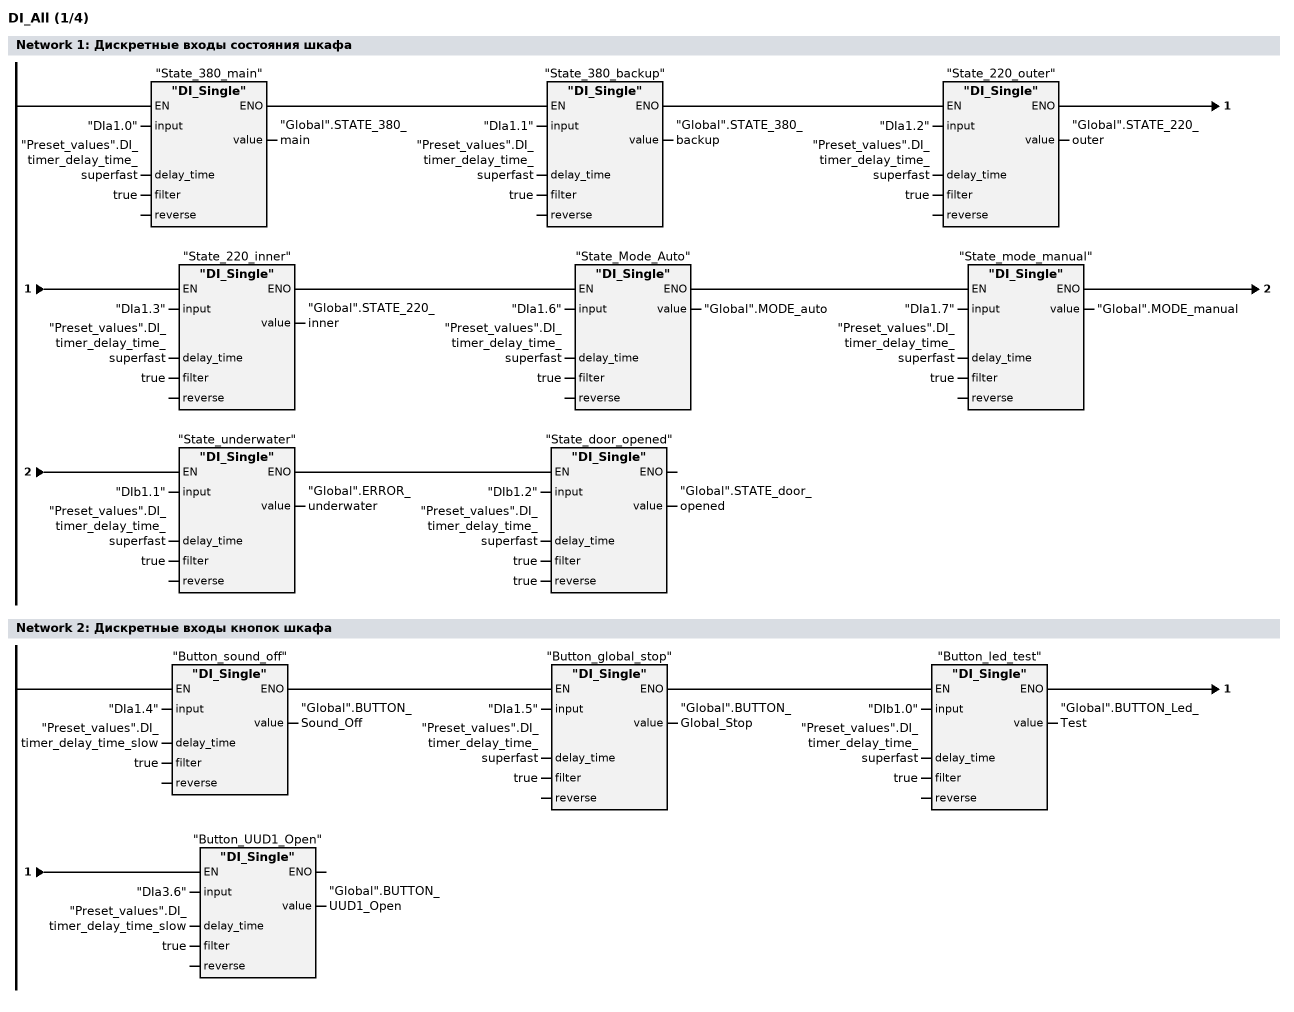
   RUNG wire#powerrail
      "State_380_main"(input := "DIa1.0", delay_time := "Preset_values".DI_timer_delay_time_superfast, filter := true, reverse :=, value => "Global".STATE_380_main)
      "State_380_backup"(input := "DIa1.1", delay_time := "Preset_values".DI_timer_delay_time_superfast, filter := true, reverse :=, value => "Global".STATE_380_backup)
      "State_220_outer"(input := "DIa1.2", delay_time := "Preset_values".DI_timer_delay_time_superfast, filter := true, reverse :=, value => "Global".STATE_220_outer)
      "State_220_inner"(input := "DIa1.3", delay_time := "Preset_values".DI_timer_delay_time_superfast, filter := true, reverse :=, value => "Global".STATE_220_inner)
      "State_Mode_Auto"(input := "DIa1.6", delay_time := "Preset_values".DI_timer_delay_time_superfast, filter := true, reverse :=, value => "Global".MODE_auto)
      "State_mode_manual"(input := "DIa1.7", delay_time := "Preset_values".DI_timer_delay_time_superfast, filter := true, reverse :=, value => "Global".MODE_manual)
      "State_underwater"(input := "DIb1.1", delay_time := "Preset_values".DI_timer_delay_time_superfast, filter := true, reverse :=, value => "Global".ERROR_underwater)
      "State_door_opened"(input := "DIb1.2", delay_time := "Preset_values".DI_timer_delay_time_superfast, filter := true, reverse := true, value => "Global".STATE_door_opened)
   END_RUNG
   // the same network as SCL:
   "State_380_main"(input := "DIa1.0",   // "DI_Single"
                    delay_time := "Preset_values".DI_timer_delay_time_superfast,
                    filter := true,
                    value => "Global".STATE_380_main,
                    ENO => #_w1);
   "State_380_backup"(EN := #_w1,   // "DI_Single"
                      input := "DIa1.1",
                      delay_time := "Preset_values".DI_timer_delay_time_superfast,
                      filter := true,
                      value => "Global".STATE_380_backup,
                      ENO => #_w2);
   "State_220_outer"(EN := #_w2,   // "DI_Single"
                     input := "DIa1.2",
                     delay_time := "Preset_values".DI_timer_delay_time_superfast,
                     filter := true,
                     value => "Global".STATE_220_outer,
                     ENO => #_w3);
   "State_220_inner"(EN := #_w3,   // "DI_Single"
                     input := "DIa1.3",
                     delay_time := "Preset_values".DI_timer_delay_time_superfast,
                     filter := true,
                     value => "Global".STATE_220_inner,
                     ENO => #_w4);
   "State_Mode_Auto"(EN := #_w4,   // "DI_Single"
                     input := "DIa1.6",
                     delay_time := "Preset_values".DI_timer_delay_time_superfast,
                     filter := true,
                     value => "Global".MODE_auto,
                     ENO => #_w5);
   "State_mode_manual"(EN := #_w5,   // "DI_Single"
                       input := "DIa1.7",
                       delay_time := "Preset_values".DI_timer_delay_time_superfast,
                       filter := true,
                       value => "Global".MODE_manual,
                       ENO => #_w6);
   "State_underwater"(EN := #_w6,   // "DI_Single"
                      input := "DIb1.1",
                      delay_time := "Preset_values".DI_timer_delay_time_superfast,
                      filter := true,
                      value => "Global".ERROR_underwater,
                      ENO => #_w7);
   IF #_w7 THEN
       "State_door_opened"(input := "DIb1.2",   // "DI_Single"
                           delay_time := "Preset_values".DI_timer_delay_time_superfast,
                           filter := true,
                           reverse := true,
                           value => "Global".STATE_door_opened);
   END_IF;
END_REGION

REGION Network 2: Дискретные входы кнопок шкафа
   RUNG wire#powerrail
      "Button_sound_off"(input := "DIa1.4", delay_time := "Preset_values".DI_timer_delay_time_slow, filter := true, reverse :=, value => "Global".BUTTON_Sound_Off)
      "Button_global_stop"(input := "DIa1.5", delay_time := "Preset_values".DI_timer_delay_time_superfast, filter := true, reverse :=, value => "Global".BUTTON_Global_Stop)
      "Button_led_test"(input := "DIb1.0", delay_time := "Preset_values".DI_timer_delay_time_superfast, filter := true, reverse :=, value => "Global".BUTTON_Led_Test)
      "Button_UUD1_Open"(input := "DIa3.6", delay_time := "Preset_values".DI_timer_delay_time_slow, filter := true, reverse :=, value => "Global".BUTTON_UUD1_Open)
   END_RUNG
   // the same network as SCL:
   "Button_sound_off"(input := "DIa1.4",   // "DI_Single"
                      delay_time := "Preset_values".DI_timer_delay_time_slow,
                      filter := true,
                      value => "Global".BUTTON_Sound_Off,
                      ENO => #_w1);
   "Button_global_stop"(EN := #_w1,   // "DI_Single"
                        input := "DIa1.5",
                        delay_time := "Preset_values".DI_timer_delay_time_superfast,
                        filter := true,
                        value => "Global".BUTTON_Global_Stop,
                        ENO => #_w2);
   "Button_led_test"(EN := #_w2,   // "DI_Single"
                     input := "DIb1.0",
                     delay_time := "Preset_values".DI_timer_delay_time_superfast,
                     filter := true,
                     value => "Global".BUTTON_Led_Test,
                     ENO => #_w3);
   IF #_w3 THEN
       "Button_UUD1_Open"(input := "DIa3.6",   // "DI_Single"
                          delay_time := "Preset_values".DI_timer_delay_time_slow,
                          filter := true,
                          value => "Global".BUTTON_UUD1_Open);
   END_IF;
END_REGION

REGION Network 3: Дискретные входы состояния насосных модулей
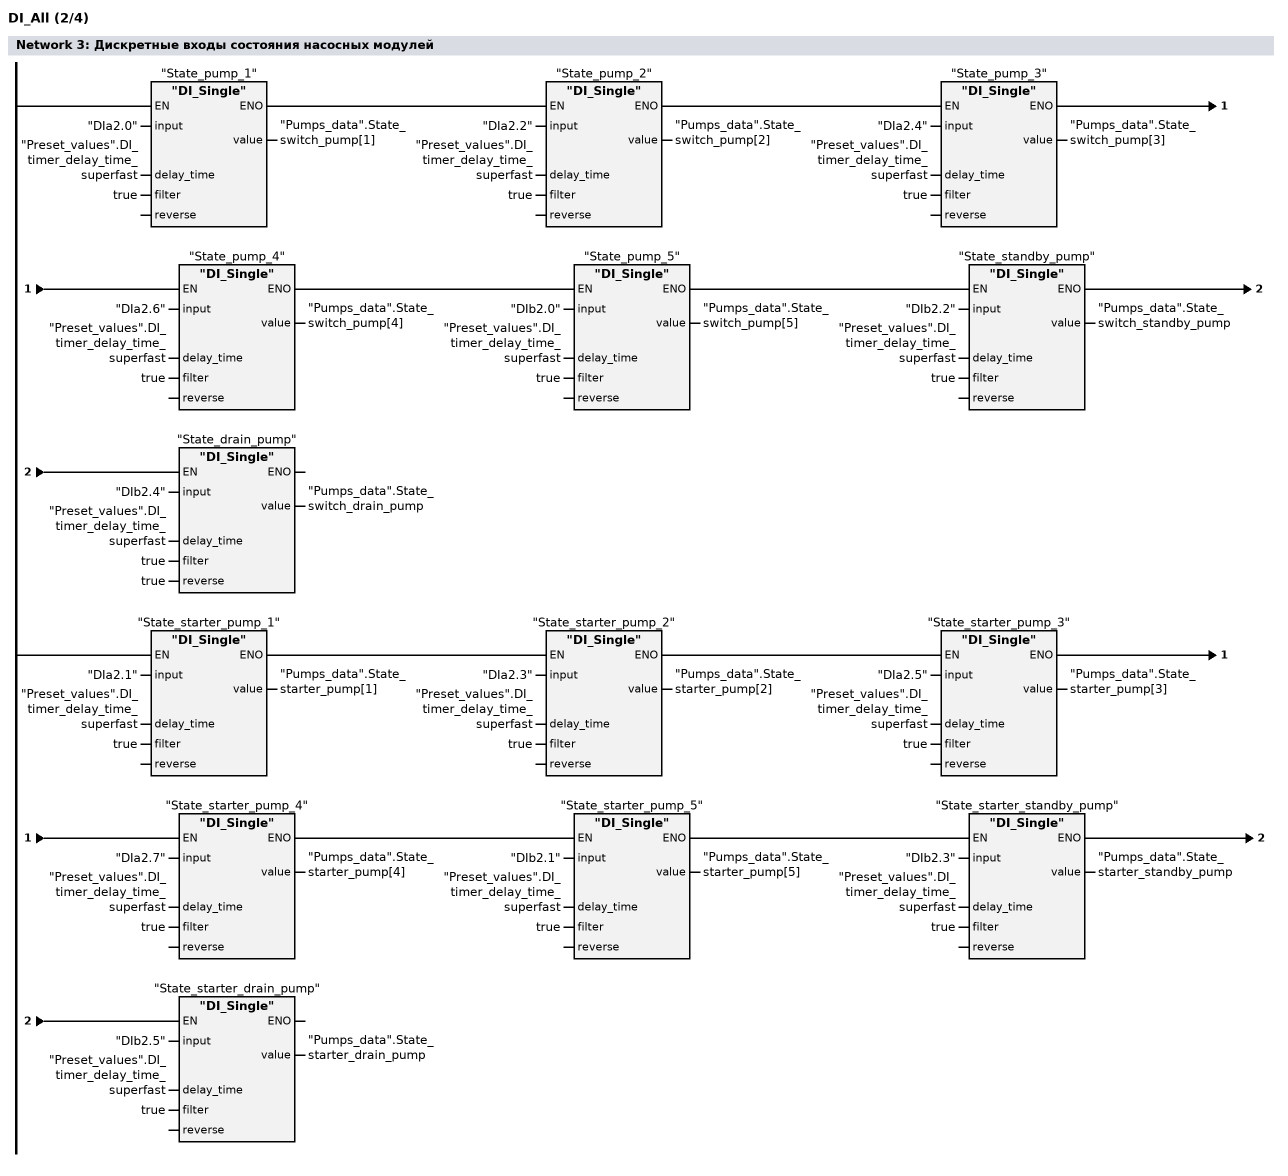
   RUNG wire#powerrail
      "State_pump_1"(input := "DIa2.0", delay_time := "Preset_values".DI_timer_delay_time_superfast, filter := true, reverse :=, value => "Pumps_data".State_switch_pump[1])
      "State_pump_2"(input := "DIa2.2", delay_time := "Preset_values".DI_timer_delay_time_superfast, filter := true, reverse :=, value => "Pumps_data".State_switch_pump[2])
      "State_pump_3"(input := "DIa2.4", delay_time := "Preset_values".DI_timer_delay_time_superfast, filter := true, reverse :=, value => "Pumps_data".State_switch_pump[3])
      "State_pump_4"(input := "DIa2.6", delay_time := "Preset_values".DI_timer_delay_time_superfast, filter := true, reverse :=, value => "Pumps_data".State_switch_pump[4])
      "State_pump_5"(input := "DIb2.0", delay_time := "Preset_values".DI_timer_delay_time_superfast, filter := true, reverse :=, value => "Pumps_data".State_switch_pump[5])
      "State_standby_pump"(input := "DIb2.2", delay_time := "Preset_values".DI_timer_delay_time_superfast, filter := true, reverse :=, value => "Pumps_data".State_switch_standby_pump)
      "State_drain_pump"(input := "DIb2.4", delay_time := "Preset_values".DI_timer_delay_time_superfast, filter := true, reverse := true, value => "Pumps_data".State_switch_drain_pump)
   END_RUNG
   RUNG wire#powerrail
      "State_starter_pump_1"(input := "DIa2.1", delay_time := "Preset_values".DI_timer_delay_time_superfast, filter := true, reverse :=, value => "Pumps_data".State_starter_pump[1])
      "State_starter_pump_2"(input := "DIa2.3", delay_time := "Preset_values".DI_timer_delay_time_superfast, filter := true, reverse :=, value => "Pumps_data".State_starter_pump[2])
      "State_starter_pump_3"(input := "DIa2.5", delay_time := "Preset_values".DI_timer_delay_time_superfast, filter := true, reverse :=, value => "Pumps_data".State_starter_pump[3])
      "State_starter_pump_4"(input := "DIa2.7", delay_time := "Preset_values".DI_timer_delay_time_superfast, filter := true, reverse :=, value => "Pumps_data".State_starter_pump[4])
      "State_starter_pump_5"(input := "DIb2.1", delay_time := "Preset_values".DI_timer_delay_time_superfast, filter := true, reverse :=, value => "Pumps_data".State_starter_pump[5])
      "State_starter_standby_pump"(input := "DIb2.3", delay_time := "Preset_values".DI_timer_delay_time_superfast, filter := true, reverse :=, value => "Pumps_data".State_starter_standby_pump)
      "State_starter_drain_pump"(input := "DIb2.5", delay_time := "Preset_values".DI_timer_delay_time_superfast, filter := true, reverse :=, value => "Pumps_data".State_starter_drain_pump)
   END_RUNG
   // the same network as SCL:
   "State_pump_1"(input := "DIa2.0",   // "DI_Single"
                  delay_time := "Preset_values".DI_timer_delay_time_superfast,
                  filter := true,
                  value => "Pumps_data".State_switch_pump[1],
                  ENO => #_w1);
   "State_pump_2"(EN := #_w1,   // "DI_Single"
                  input := "DIa2.2",
                  delay_time := "Preset_values".DI_timer_delay_time_superfast,
                  filter := true,
                  value => "Pumps_data".State_switch_pump[2],
                  ENO => #_w2);
   "State_pump_3"(EN := #_w2,   // "DI_Single"
                  input := "DIa2.4",
                  delay_time := "Preset_values".DI_timer_delay_time_superfast,
                  filter := true,
                  value => "Pumps_data".State_switch_pump[3],
                  ENO => #_w3);
   "State_pump_4"(EN := #_w3,   // "DI_Single"
                  input := "DIa2.6",
                  delay_time := "Preset_values".DI_timer_delay_time_superfast,
                  filter := true,
                  value => "Pumps_data".State_switch_pump[4],
                  ENO => #_w4);
   "State_pump_5"(EN := #_w4,   // "DI_Single"
                  input := "DIb2.0",
                  delay_time := "Preset_values".DI_timer_delay_time_superfast,
                  filter := true,
                  value => "Pumps_data".State_switch_pump[5],
                  ENO => #_w5);
   "State_standby_pump"(EN := #_w5,   // "DI_Single"
                        input := "DIb2.2",
                        delay_time := "Preset_values".DI_timer_delay_time_superfast,
                        filter := true,
                        value => "Pumps_data".State_switch_standby_pump,
                        ENO => #_w6);
   IF #_w6 THEN
       "State_drain_pump"(input := "DIb2.4",   // "DI_Single"
                          delay_time := "Preset_values".DI_timer_delay_time_superfast,
                          filter := true,
                          reverse := true,
                          value => "Pumps_data".State_switch_drain_pump);
   END_IF;
   "State_starter_pump_1"(input := "DIa2.1",   // "DI_Single"
                          delay_time := "Preset_values".DI_timer_delay_time_superfast,
                          filter := true,
                          value => "Pumps_data".State_starter_pump[1],
                          ENO => #_w7);
   "State_starter_pump_2"(EN := #_w7,   // "DI_Single"
                          input := "DIa2.3",
                          delay_time := "Preset_values".DI_timer_delay_time_superfast,
                          filter := true,
                          value => "Pumps_data".State_starter_pump[2],
                          ENO => #_w8);
   "State_starter_pump_3"(EN := #_w8,   // "DI_Single"
                          input := "DIa2.5",
                          delay_time := "Preset_values".DI_timer_delay_time_superfast,
                          filter := true,
                          value => "Pumps_data".State_starter_pump[3],
                          ENO => #_w9);
   "State_starter_pump_4"(EN := #_w9,   // "DI_Single"
                          input := "DIa2.7",
                          delay_time := "Preset_values".DI_timer_delay_time_superfast,
                          filter := true,
                          value => "Pumps_data".State_starter_pump[4],
                          ENO => #_w10);
   "State_starter_pump_5"(EN := #_w10,   // "DI_Single"
                          input := "DIb2.1",
                          delay_time := "Preset_values".DI_timer_delay_time_superfast,
                          filter := true,
                          value => "Pumps_data".State_starter_pump[5],
                          ENO => #_w11);
   "State_starter_standby_pump"(EN := #_w11,   // "DI_Single"
                           input := "DIb2.3",
                           delay_time := "Preset_values".DI_timer_delay_time_superfast,
                           filter := true,
                           value => "Pumps_data".State_starter_standby_pump,
                           ENO => #_w12);
   IF #_w12 THEN
       "State_starter_drain_pump"(input := "DIb2.5",   // "DI_Single"
                               delay_time := "Preset_values".DI_timer_delay_time_superfast,
                               filter := true,
                               value => "Pumps_data".State_starter_drain_pump);
   END_IF;
END_REGION

REGION Network 4: Дискретные входы протоков УУС
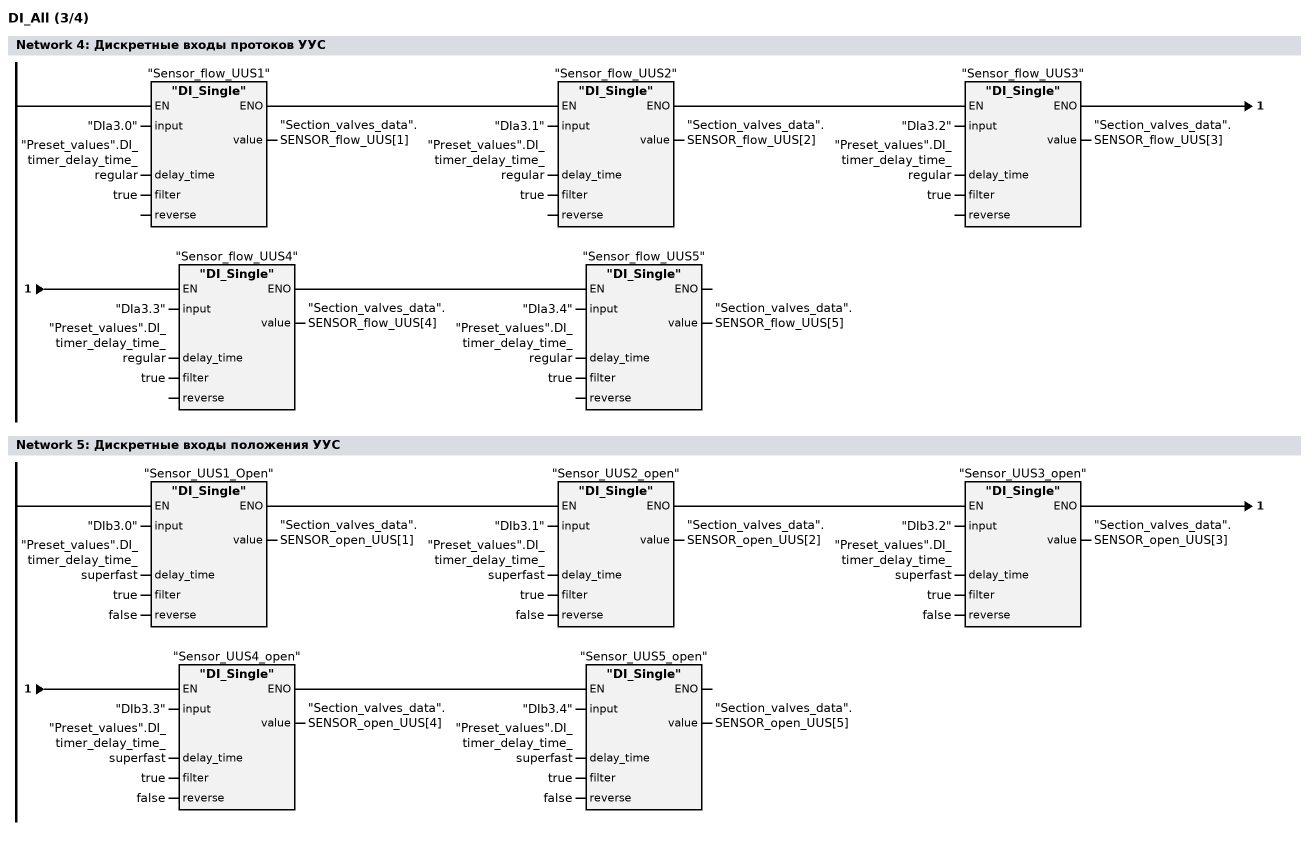
   RUNG wire#powerrail
      "Sensor_flow_UUS1"(input := "DIa3.0", delay_time := "Preset_values".DI_timer_delay_time_regular, filter := true, reverse :=, value => "Section_valves_data".SENSOR_flow_UUS[1])
      "Sensor_flow_UUS2"(input := "DIa3.1", delay_time := "Preset_values".DI_timer_delay_time_regular, filter := true, reverse :=, value => "Section_valves_data".SENSOR_flow_UUS[2])
      "Sensor_flow_UUS3"(input := "DIa3.2", delay_time := "Preset_values".DI_timer_delay_time_regular, filter := true, reverse :=, value => "Section_valves_data".SENSOR_flow_UUS[3])
      "Sensor_flow_UUS4"(input := "DIa3.3", delay_time := "Preset_values".DI_timer_delay_time_regular, filter := true, reverse :=, value => "Section_valves_data".SENSOR_flow_UUS[4])
      "Sensor_flow_UUS5"(input := "DIa3.4", delay_time := "Preset_values".DI_timer_delay_time_regular, filter := true, reverse :=, value => "Section_valves_data".SENSOR_flow_UUS[5])
   END_RUNG
   // the same network as SCL:
   "Sensor_flow_UUS1"(input := "DIa3.0",   // "DI_Single"
                      delay_time := "Preset_values".DI_timer_delay_time_regular,
                      filter := true,
                      value => "Section_valves_data".SENSOR_flow_UUS[1],
                      ENO => #_w1);
   "Sensor_flow_UUS2"(EN := #_w1,   // "DI_Single"
                      input := "DIa3.1",
                      delay_time := "Preset_values".DI_timer_delay_time_regular,
                      filter := true,
                      value => "Section_valves_data".SENSOR_flow_UUS[2],
                      ENO => #_w2);
   "Sensor_flow_UUS3"(EN := #_w2,   // "DI_Single"
                      input := "DIa3.2",
                      delay_time := "Preset_values".DI_timer_delay_time_regular,
                      filter := true,
                      value => "Section_valves_data".SENSOR_flow_UUS[3],
                      ENO => #_w3);
   "Sensor_flow_UUS4"(EN := #_w3,   // "DI_Single"
                      input := "DIa3.3",
                      delay_time := "Preset_values".DI_timer_delay_time_regular,
                      filter := true,
                      value => "Section_valves_data".SENSOR_flow_UUS[4],
                      ENO => #_w4);
   IF #_w4 THEN
       "Sensor_flow_UUS5"(input := "DIa3.4",   // "DI_Single"
                          delay_time := "Preset_values".DI_timer_delay_time_regular,
                          filter := true,
                          value => "Section_valves_data".SENSOR_flow_UUS[5]);
   END_IF;
END_REGION

REGION Network 5: Дискретные входы положения УУС
   RUNG wire#powerrail
      "Sensor_UUS1_Open"(input := "DIb3.0", delay_time := "Preset_values".DI_timer_delay_time_superfast, filter := true, reverse := false, value => "Section_valves_data".SENSOR_open_UUS[1])
      "Sensor_UUS2_open"(input := "DIb3.1", delay_time := "Preset_values".DI_timer_delay_time_superfast, filter := true, reverse := false, value => "Section_valves_data".SENSOR_open_UUS[2])
      "Sensor_UUS3_open"(input := "DIb3.2", delay_time := "Preset_values".DI_timer_delay_time_superfast, filter := true, reverse := false, value => "Section_valves_data".SENSOR_open_UUS[3])
      "Sensor_UUS4_open"(input := "DIb3.3", delay_time := "Preset_values".DI_timer_delay_time_superfast, filter := true, reverse := false, value => "Section_valves_data".SENSOR_open_UUS[4])
      "Sensor_UUS5_open"(input := "DIb3.4", delay_time := "Preset_values".DI_timer_delay_time_superfast, filter := true, reverse := false, value => "Section_valves_data".SENSOR_open_UUS[5])
   END_RUNG
   // the same network as SCL:
   "Sensor_UUS1_Open"(input := "DIb3.0",   // "DI_Single"
                      delay_time := "Preset_values".DI_timer_delay_time_superfast,
                      filter := true,
                      reverse := false,
                      value => "Section_valves_data".SENSOR_open_UUS[1],
                      ENO => #_w1);
   "Sensor_UUS2_open"(EN := #_w1,   // "DI_Single"
                      input := "DIb3.1",
                      delay_time := "Preset_values".DI_timer_delay_time_superfast,
                      filter := true,
                      reverse := false,
                      value => "Section_valves_data".SENSOR_open_UUS[2],
                      ENO => #_w2);
   "Sensor_UUS3_open"(EN := #_w2,   // "DI_Single"
                      input := "DIb3.2",
                      delay_time := "Preset_values".DI_timer_delay_time_superfast,
                      filter := true,
                      reverse := false,
                      value => "Section_valves_data".SENSOR_open_UUS[3],
                      ENO => #_w3);
   "Sensor_UUS4_open"(EN := #_w3,   // "DI_Single"
                      input := "DIb3.3",
                      delay_time := "Preset_values".DI_timer_delay_time_superfast,
                      filter := true,
                      reverse := false,
                      value => "Section_valves_data".SENSOR_open_UUS[4],
                      ENO => #_w4);
   IF #_w4 THEN
       "Sensor_UUS5_open"(input := "DIb3.4",   // "DI_Single"
                          delay_time := "Preset_values".DI_timer_delay_time_superfast,
                          filter := true,
                          reverse := false,
                          value => "Section_valves_data".SENSOR_open_UUS[5]);
   END_IF;
END_REGION

REGION Network 6: Дискретные входы положения шаровых кранов
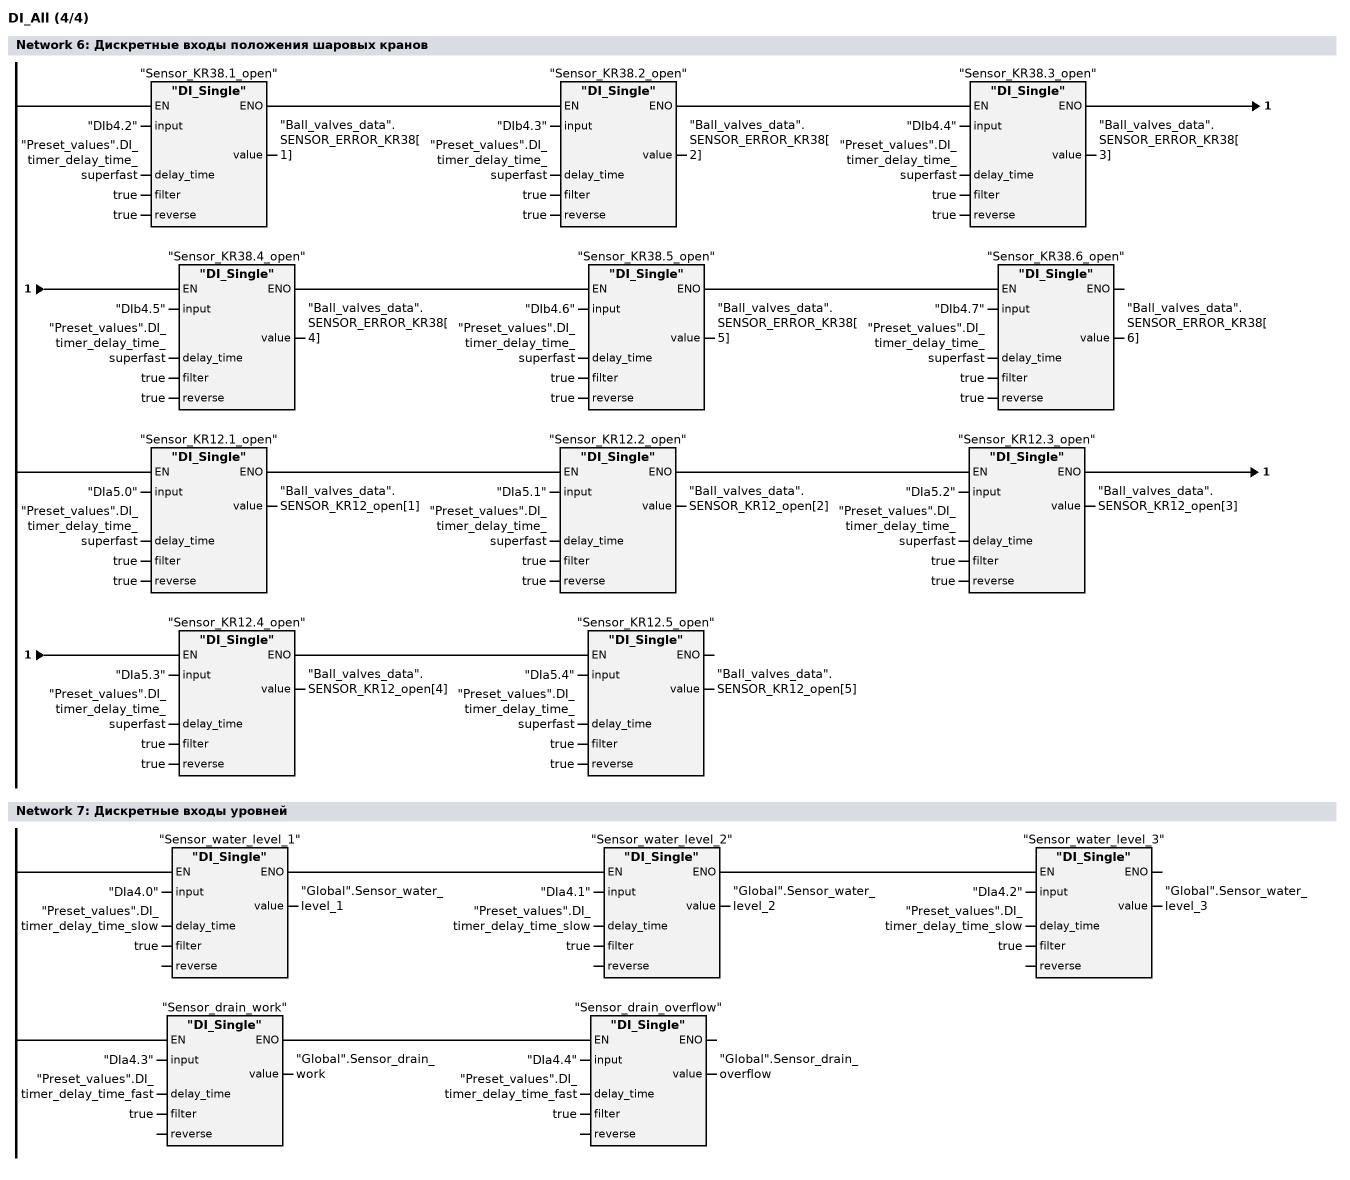
   RUNG wire#powerrail
      "Sensor_KR38.1_open"(input := "DIb4.2", delay_time := "Preset_values".DI_timer_delay_time_superfast, filter := true, reverse := true, value => "Ball_valves_data".SENSOR_ERROR_KR38[1])
      "Sensor_KR38.2_open"(input := "DIb4.3", delay_time := "Preset_values".DI_timer_delay_time_superfast, filter := true, reverse := true, value => "Ball_valves_data".SENSOR_ERROR_KR38[2])
      "Sensor_KR38.3_open"(input := "DIb4.4", delay_time := "Preset_values".DI_timer_delay_time_superfast, filter := true, reverse := true, value => "Ball_valves_data".SENSOR_ERROR_KR38[3])
      "Sensor_KR38.4_open"(input := "DIb4.5", delay_time := "Preset_values".DI_timer_delay_time_superfast, filter := true, reverse := true, value => "Ball_valves_data".SENSOR_ERROR_KR38[4])
      "Sensor_KR38.5_open"(input := "DIb4.6", delay_time := "Preset_values".DI_timer_delay_time_superfast, filter := true, reverse := true, value => "Ball_valves_data".SENSOR_ERROR_KR38[5])
      "Sensor_KR38.6_open"(input := "DIb4.7", delay_time := "Preset_values".DI_timer_delay_time_superfast, filter := true, reverse := true, value => "Ball_valves_data".SENSOR_ERROR_KR38[6])
   END_RUNG
   RUNG wire#powerrail
      "Sensor_KR12.1_open"(input := "DIa5.0", delay_time := "Preset_values".DI_timer_delay_time_superfast, filter := true, reverse := true, value => "Ball_valves_data".SENSOR_KR12_open[1])
      "Sensor_KR12.2_open"(input := "DIa5.1", delay_time := "Preset_values".DI_timer_delay_time_superfast, filter := true, reverse := true, value => "Ball_valves_data".SENSOR_KR12_open[2])
      "Sensor_KR12.3_open"(input := "DIa5.2", delay_time := "Preset_values".DI_timer_delay_time_superfast, filter := true, reverse := true, value => "Ball_valves_data".SENSOR_KR12_open[3])
      "Sensor_KR12.4_open"(input := "DIa5.3", delay_time := "Preset_values".DI_timer_delay_time_superfast, filter := true, reverse := true, value => "Ball_valves_data".SENSOR_KR12_open[4])
      "Sensor_KR12.5_open"(input := "DIa5.4", delay_time := "Preset_values".DI_timer_delay_time_superfast, filter := true, reverse := true, value => "Ball_valves_data".SENSOR_KR12_open[5])
   END_RUNG
   // the same network as SCL:
   "Sensor_KR38.1_open"(input := "DIb4.2",   // "DI_Single"
                        delay_time := "Preset_values".DI_timer_delay_time_superfast,
                        filter := true,
                        reverse := true,
                        value => "Ball_valves_data".SENSOR_ERROR_KR38[1],
                        ENO => #_w1);
   "Sensor_KR38.2_open"(EN := #_w1,   // "DI_Single"
                        input := "DIb4.3",
                        delay_time := "Preset_values".DI_timer_delay_time_superfast,
                        filter := true,
                        reverse := true,
                        value => "Ball_valves_data".SENSOR_ERROR_KR38[2],
                        ENO => #_w2);
   "Sensor_KR38.3_open"(EN := #_w2,   // "DI_Single"
                        input := "DIb4.4",
                        delay_time := "Preset_values".DI_timer_delay_time_superfast,
                        filter := true,
                        reverse := true,
                        value => "Ball_valves_data".SENSOR_ERROR_KR38[3],
                        ENO => #_w3);
   "Sensor_KR38.4_open"(EN := #_w3,   // "DI_Single"
                        input := "DIb4.5",
                        delay_time := "Preset_values".DI_timer_delay_time_superfast,
                        filter := true,
                        reverse := true,
                        value => "Ball_valves_data".SENSOR_ERROR_KR38[4],
                        ENO => #_w4);
   "Sensor_KR38.5_open"(EN := #_w4,   // "DI_Single"
                        input := "DIb4.6",
                        delay_time := "Preset_values".DI_timer_delay_time_superfast,
                        filter := true,
                        reverse := true,
                        value => "Ball_valves_data".SENSOR_ERROR_KR38[5],
                        ENO => #_w5);
   IF #_w5 THEN
       "Sensor_KR38.6_open"(input := "DIb4.7",   // "DI_Single"
                            delay_time := "Preset_values".DI_timer_delay_time_superfast,
                            filter := true,
                            reverse := true,
                            value => "Ball_valves_data".SENSOR_ERROR_KR38[6]);
   END_IF;
   "Sensor_KR12.1_open"(input := "DIa5.0",   // "DI_Single"
                        delay_time := "Preset_values".DI_timer_delay_time_superfast,
                        filter := true,
                        reverse := true,
                        value => "Ball_valves_data".SENSOR_KR12_open[1],
                        ENO => #_w6);
   "Sensor_KR12.2_open"(EN := #_w6,   // "DI_Single"
                        input := "DIa5.1",
                        delay_time := "Preset_values".DI_timer_delay_time_superfast,
                        filter := true,
                        reverse := true,
                        value => "Ball_valves_data".SENSOR_KR12_open[2],
                        ENO => #_w7);
   "Sensor_KR12.3_open"(EN := #_w7,   // "DI_Single"
                        input := "DIa5.2",
                        delay_time := "Preset_values".DI_timer_delay_time_superfast,
                        filter := true,
                        reverse := true,
                        value => "Ball_valves_data".SENSOR_KR12_open[3],
                        ENO => #_w8);
   "Sensor_KR12.4_open"(EN := #_w8,   // "DI_Single"
                        input := "DIa5.3",
                        delay_time := "Preset_values".DI_timer_delay_time_superfast,
                        filter := true,
                        reverse := true,
                        value => "Ball_valves_data".SENSOR_KR12_open[4],
                        ENO => #_w9);
   IF #_w9 THEN
       "Sensor_KR12.5_open"(input := "DIa5.4",   // "DI_Single"
                            delay_time := "Preset_values".DI_timer_delay_time_superfast,
                            filter := true,
                            reverse := true,
                            value => "Ball_valves_data".SENSOR_KR12_open[5]);
   END_IF;
END_REGION

REGION Network 7: Дискретные входы уровней
   RUNG wire#powerrail
      "Sensor_water_level_1"(input := "DIa4.0", delay_time := "Preset_values".DI_timer_delay_time_slow, filter := true, reverse :=, value => "Global".Sensor_water_level_1)
      "Sensor_water_level_2"(input := "DIa4.1", delay_time := "Preset_values".DI_timer_delay_time_slow, filter := true, reverse :=, value => "Global".Sensor_water_level_2)
      "Sensor_water_level_3"(input := "DIa4.2", delay_time := "Preset_values".DI_timer_delay_time_slow, filter := true, reverse :=, value => "Global".Sensor_water_level_3)
   END_RUNG
   RUNG wire#powerrail
      "Sensor_drain_work"(input := "DIa4.3", delay_time := "Preset_values".DI_timer_delay_time_fast, filter := true, reverse :=, value => "Global".Sensor_drain_work)
      "Sensor_drain_overflow"(input := "DIa4.4", delay_time := "Preset_values".DI_timer_delay_time_fast, filter := true, reverse :=, value => "Global".Sensor_drain_overflow)
   END_RUNG
   // the same network as SCL:
   "Sensor_water_level_1"(input := "DIa4.0",   // "DI_Single"
                          delay_time := "Preset_values".DI_timer_delay_time_slow,
                          filter := true,
                          value => "Global".Sensor_water_level_1,
                          ENO => #_w1);
   "Sensor_water_level_2"(EN := #_w1,   // "DI_Single"
                          input := "DIa4.1",
                          delay_time := "Preset_values".DI_timer_delay_time_slow,
                          filter := true,
                          value => "Global".Sensor_water_level_2,
                          ENO => #_w2);
   IF #_w2 THEN
       "Sensor_water_level_3"(input := "DIa4.2",   // "DI_Single"
                              delay_time := "Preset_values".DI_timer_delay_time_slow,
                              filter := true,
                              value => "Global".Sensor_water_level_3);
   END_IF;
   "Sensor_drain_work"(input := "DIa4.3",   // "DI_Single"
                       delay_time := "Preset_values".DI_timer_delay_time_fast,
                       filter := true,
                       value => "Global".Sensor_drain_work,
                       ENO => #_w3);
   IF #_w3 THEN
       "Sensor_drain_overflow"(input := "DIa4.4",   // "DI_Single"
                               delay_time := "Preset_values".DI_timer_delay_time_fast,
                               filter := true,
                               value => "Global".Sensor_drain_overflow);
   END_IF;
END_REGION
END_FUNCTION

FUNCTION "AI_All" : Void   // FC2, LAD
{ S7_Optimized_Access := 'TRUE' }
VERSION : 0.1
   VAR_TEMP   // added for the SCL form of the ladder/FBD networks
      _w1 : Bool;
      _w2 : Bool;
      _w3 : Bool;
      _w4 : Bool;
      _w5 : Bool;
      _w6 : Bool;
      _w7 : Bool;
   END_VAR
BEGIN

